gfCNCPoint5[10865] = {X 236.2309, Y 48.3200, Z -7.1667, A 0.000, B 0.000, C 0.000 }
gfCNCPoint5[10866] = {X 235.6245, Y 47.5134, Z -7.1667, A 0.000, B 0.000, C 0.000 }
gfCNCPoint5[10867] = {X 235.1970, Y 46.5992, Z -7.1667, A 0.000, B 0.000, C 0.000 }
gfCNCPoint5[10868] = {X 234.9666, Y 45.6167, Z -7.1667, A 0.000, B 0.000, C 0.000 }
gfCNCPoint5[10869] = {X 234.9373, Y 45.3090, Z -7.1667, A 0.000, B 0.000, C 0.000 }
gfCNCPoint5[10870] = {X 234.9275, Y 45.0000, Z -7.1667, A 0.000, B 0.000, C 0.000 }
gfCNCPoint5[10871] = {X 234.9275, Y 44.2089, Z -7.1667, A 0.000, B 0.000, C 0.000 }
gfCNCPoint5[10872] = {X 235.0194, Y 43.2661, Z -7.1667, A 0.000, B 0.000, C 0.000 }
gfCNCPoint5[10873] = {X 235.2918, Y 42.3588, Z -7.1667, A 0.000, B 0.000, C 0.000 }
gfCNCPoint5[10874] = {X 235.7342, Y 41.5212, Z -7.1667, A 0.000, B 0.000, C 0.000 }
gfCNCPoint5[10875] = {X 236.3302, Y 40.7849, Z -7.1667, A 0.000, B 0.000, C 0.000 }
gfCNCPoint5[10876] = {X 237.0572, Y 40.1776, Z -7.1667, A 0.000, B 0.000, C 0.000 }
gfCNCPoint5[10877] = {X 237.8878, Y 39.7222, Z -7.1667, A 0.000, B 0.000, C 0.000 }
gfCNCPoint5[10878] = {X 241.5460, Y 32.5618, Z -7.1667, A 0.000, B 0.000, C 0.000 }
gfCNCPoint5[10879] = {X 240.2114, Y 31.5589, Z -7.1667, A 0.000, B 0.000, C 0.000 }
gfCNCPoint5[10880] = {X 239.0306, Y 30.3788, Z -7.1667, A 0.000, B 0.000, C 0.000 }
gfCNCPoint5[10881] = {X 238.0268, Y 29.0450, Z -7.1667, A 0.000, B 0.000, C 0.000 }
gfCNCPoint5[10882] = {X 237.2198, Y 27.5836, Z -7.1667, A 0.000, B 0.000, C 0.000 }
gfCNCPoint5[10883] = {X 236.6256, Y 26.0236, Z -7.1667, A 0.000, B 0.000, C 0.000 }
gfCNCPoint5[10884] = {X 236.1904, Y 24.1499, Z -7.1667, A 0.000, B 0.000, C 0.000 }
gfCNCPoint5[10885] = {X 235.9685, Y 22.2393, Z -7.1667, A 0.000, B 0.000, C 0.000 }
gfCNCPoint5[10886] = {X 235.9626, Y 20.3158, Z -7.1667, A 0.000, B 0.000, C 0.000 }
gfCNCPoint5[10887] = {X 236.1729, Y 18.4038, Z -7.1667, A 0.000, B 0.000, C 0.000 }
gfCNCPoint5[10888] = {X 236.5966, Y 16.5276, Z -7.1667, A 0.000, B 0.000, C 0.000 }
gfCNCPoint5[10889] = {X 237.1160, Y 15.0570, Z -7.1667, A 0.000, B 0.000, C 0.000 }
gfCNCPoint5[10890] = {X 237.8157, Y 13.6631, Z -7.1667, A 0.000, B 0.000, C 0.000 }
gfCNCPoint5[10891] = {X 238.6848, Y 12.3680, Z -7.1667, A 0.000, B 0.000, C 0.000 }
gfCNCPoint5[10892] = {X 239.7094, Y 11.1921, Z -7.1667, A 0.000, B 0.000, C 0.000 }
gfCNCPoint5[10893] = {X 240.8738, Y 10.1538, Z -7.1667, A 0.000, B 0.000, C 0.000 }
gfCNCPoint5[10894] = {X 242.1593, Y 9.2697, Z -7.1667, A 0.000, B 0.000, C 0.000 }
gfCNCPoint5[10895] = {X 243.5456, Y 8.5539, Z -7.1667, A 0.000, B 0.000, C 0.000 }
gfCNCPoint5[10896] = {X 245.0107, Y 8.0176, Z -7.1667, A 0.000, B 0.000, C 0.000 }
gfCNCPoint5[10897] = {X 246.5316, Y 7.6695, Z -7.1667, A 0.000, B 0.000, C 0.000 }
gfCNCPoint5[10898] = {X 248.6761, Y 7.3920, Z -7.1667, A 0.000, B 0.000, C 0.000 }
gfCNCPoint5[10899] = {X 250.8369, Y 7.3096, Z -7.1667, A 0.000, B 0.000, C 0.000 }
gfCNCPoint5[10900] = {X 266.7608, Y 7.3096, Z -7.1667, A 0.000, B 0.000, C 0.000 }
gfCNCPoint5[10901] = {X 267.7192, Y 7.4110, Z -7.1667, A 0.000, B 0.000, C 0.000 }
gfCNCPoint5[10902] = {X 268.6390, Y 7.6987, Z -7.1667, A 0.000, B 0.000, C 0.000 }
gfCNCPoint5[10903] = {X 269.4844, Y 8.1615, Z -7.1667, A 0.000, B 0.000, C 0.000 }
gfCNCPoint5[10904] = {X 270.2224, Y 8.7814, Z -7.1667, A 0.000, B 0.000, C 0.000 }
gfCNCPoint5[10905] = {X 270.8243, Y 9.5341, Z -7.1667, A 0.000, B 0.000, C 0.000 }
gfCNCPoint5[10906] = {X 271.2665, Y 10.3904, Z -7.1667, A 0.000, B 0.000, C 0.000 }
gfCNCPoint5[10907] = {X 271.5236, Y 11.2718, Z -7.1667, A 0.000, B 0.000, C 0.000 }
gfCNCPoint5[10908] = {X 271.6110, Y 12.1858, Z -7.1667, A 0.000, B 0.000, C 0.000 }
gfCNCPoint5[10909] = {X 271.6108, Y 13.0237, Z -7.1667, A 0.000, B 0.000, C 0.000 }
gfCNCPoint5[10910] = {X 271.5128, Y 13.9524, Z -7.1667, A 0.000, B 0.000, C 0.000 }
gfCNCPoint5[10911] = {X 271.2396, Y 14.8453, Z -7.1667, A 0.000, B 0.000, C 0.000 }
gfCNCPoint5[10912] = {X 275.6743, Y 16.6820, Z -7.1667, A 0.000, B 0.000, C 0.000 }
gfCNCPoint5[10913] = {X 275.3129, Y 17.4561, Z -7.1667, A 0.000, B 0.000, C 0.000 }
gfCNCPoint5[10914] = {X 274.8847, Y 18.1954, Z -7.1667, A 0.000, B 0.000, C 0.000 }
gfCNCPoint5[10915] = {X 274.8848, Y 38.9916, Z -7.1667, A 0.000, B 0.000, C 0.000 }
gfCNCPoint5[10916] = {X 275.3141, Y 39.7329, Z -7.1667, A 0.000, B 0.000, C 0.000 }
gfCNCPoint5[10917] = {X 275.6762, Y 40.5092, Z -7.1667, A 0.000, B 0.000, C 0.000 }
gfCNCPoint5[10918] = {X 276.0370, Y 39.7351, Z -7.1667, A 0.000, B 0.000, C 0.000 }
gfCNCPoint5[10919] = {X 276.4644, Y 38.9955, Z -7.1667, A 0.000, B 0.000, C 0.000 }
gfCNCPoint5[10920] = {X 276.4643, Y 18.1958, Z -7.1667, A 0.000, B 0.000, C 0.000 }
gfCNCPoint5[10921] = {X 276.0359, Y 17.4563, Z -7.1667, A 0.000, B 0.000, C 0.000 }
gfCNCPoint5[10922] = {X 275.6743, Y 16.6820, Z -7.1667, A 0.000, B 0.000, C 0.000 }
gfCNCPoint5[10923] = {X 273.4570, Y 15.7637, Z -7.1667, A 0.000, B 0.000, C 0.000 }
gfCNCPoint5[10924] = {X 273.0268, Y 16.6335, Z -7.1667, A 0.000, B 0.000, C 0.000 }
gfCNCPoint5[10925] = {X 272.4847, Y 17.4383, Z -7.1667, A 0.000, B 0.000, C 0.000 }
gfCNCPoint5[10926] = {X 272.4848, Y 39.7486, Z -7.1667, A 0.000, B 0.000, C 0.000 }
gfCNCPoint5[10927] = {X 273.0277, Y 40.5550, Z -7.1667, A 0.000, B 0.000, C 0.000 }
gfCNCPoint5[10928] = {X 273.4584, Y 41.4265, Z -7.1667, A 0.000, B 0.000, C 0.000 }
gfCNCPoint5[10929] = {X 273.7587, Y 42.3088, Z -7.1667, A 0.000, B 0.000, C 0.000 }
gfCNCPoint5[10930] = {X 273.9439, Y 43.2222, Z -7.1667, A 0.000, B 0.000, C 0.000 }
gfCNCPoint5[10931] = {X 274.0108, Y 44.1519, Z -7.1667, A 0.000, B 0.000, C 0.000 }
gfCNCPoint5[10932] = {X 274.0110, Y 45.0000, Z -7.1667, A 0.000, B 0.000, C 0.000 }
gfCNCPoint5[10933] = {X 273.9884, Y 45.5734, Z -7.1667, A 0.000, B 0.000, C 0.000 }
gfCNCPoint5[10934] = {X 273.9207, Y 46.1433, Z -7.1667, A 0.000, B 0.000, C 0.000 }
gfCNCPoint5[10935] = {X 275.0713, Y 45.9760, Z -7.1667, A 0.000, B 0.000, C 0.000 }
gfCNCPoint5[10936] = {X 276.2327, Y 45.9200, Z -7.1667, A 0.000, B 0.000, C 0.000 }
gfCNCPoint5[10937] = {X 277.3960, Y 45.9200, Z -7.1667, A 0.000, B 0.000, C 0.000 }
gfCNCPoint5[10938] = {X 277.3539, Y 45.4858, Z -7.1667, A 0.000, B 0.000, C 0.000 }
gfCNCPoint5[10939] = {X 277.3378, Y 45.0498, Z -7.1667, A 0.000, B 0.000, C 0.000 }
gfCNCPoint5[10940] = {X 277.3377, Y 44.2000, Z -7.1667, A 0.000, B 0.000, C 0.000 }
gfCNCPoint5[10941] = {X 277.4025, Y 43.2541, Z -7.1667, A 0.000, B 0.000, C 0.000 }
gfCNCPoint5[10942] = {X 277.5889, Y 42.3244, Z -7.1667, A 0.000, B 0.000, C 0.000 }
gfCNCPoint5[10943] = {X 277.8939, Y 41.4266, Z -7.1667, A 0.000, B 0.000, C 0.000 }
gfCNCPoint5[10944] = {X 278.3235, Y 40.5564, Z -7.1667, A 0.000, B 0.000, C 0.000 }
gfCNCPoint5[10945] = {X 278.8644, Y 39.7505, Z -7.1667, A 0.000, B 0.000, C 0.000 }
gfCNCPoint5[10946] = {X 278.8643, Y 17.4386, Z -7.1667, A 0.000, B 0.000, C 0.000 }
gfCNCPoint5[10947] = {X 278.3220, Y 16.6336, Z -7.1667, A 0.000, B 0.000, C 0.000 }
gfCNCPoint5[10948] = {X 277.8917, Y 15.7637, Z -7.1667, A 0.000, B 0.000, C 0.000 }
gfCNCPoint5[10949] = {X 277.5902, Y 14.8788, Z -7.1667, A 0.000, B 0.000, C 0.000 }
gfCNCPoint5[10950] = {X 277.4046, Y 13.9627, Z -7.1667, A 0.000, B 0.000, C 0.000 }
gfCNCPoint5[10951] = {X 277.3379, Y 13.0303, Z -7.1667, A 0.000, B 0.000, C 0.000 }
gfCNCPoint5[10952] = {X 277.3377, Y 12.1868, Z -7.1667, A 0.000, B 0.000, C 0.000 }
gfCNCPoint5[10953] = {X 277.3952, Y 11.2737, Z -7.1667, A 0.000, B 0.000, C 0.000 }
gfCNCPoint5[10954] = {X 277.5667, Y 10.3750, Z -7.1667, A 0.000, B 0.000, C 0.000 }
gfCNCPoint5[10955] = {X 277.8497, Y 9.5049, Z -7.1667, A 0.000, B 0.000, C 0.000 }
gfCNCPoint5[10956] = {X 273.4972, Y 9.5049, Z -7.1667, A 0.000, B 0.000, C 0.000 }
gfCNCPoint5[10957] = {X 273.7804, Y 10.3736, Z -7.1667, A 0.000, B 0.000, C 0.000 }
gfCNCPoint5[10958] = {X 273.9526, Y 11.2709, Z -7.1667, A 0.000, B 0.000, C 0.000 }
gfCNCPoint5[10959] = {X 274.0110, Y 12.1828, Z -7.1667, A 0.000, B 0.000, C 0.000 }
gfCNCPoint5[10960] = {X 274.0107, Y 13.0462, Z -7.1667, A 0.000, B 0.000, C 0.000 }
gfCNCPoint5[10961] = {X 273.9427, Y 13.9732, Z -7.1667, A 0.000, B 0.000, C 0.000 }
gfCNCPoint5[10962] = {X 273.7571, Y 14.8840, Z -7.1667, A 0.000, B 0.000, C 0.000 }
gfCNCPoint5[10963] = {X 273.4570, Y 15.7637, Z -7.1667, A 0.000, B 0.000, C 0.000 }
gfCNCPoint5[10964] = {X 271.2396, Y 14.8453, Z -7.1667, A 0.000, B 0.000, C 0.000 }
gfCNCPoint5[10965] = {X 270.7507, Y 15.7451, Z -7.1667, A 0.000, B 0.000, C 0.000 }
gfCNCPoint5[10966] = {X 270.0847, Y 16.5231, Z -7.1667, A 0.000, B 0.000, C 0.000 }
gfCNCPoint5[10967] = {X 270.0848, Y 40.6638, Z -7.1667, A 0.000, B 0.000, C 0.000 }
gfCNCPoint5[10968] = {X 270.7249, Y 41.4045, Z -7.1667, A 0.000, B 0.000, C 0.000 }
gfCNCPoint5[10969] = {X 271.2042, Y 42.2581, Z -7.1667, A 0.000, B 0.000, C 0.000 }
gfCNCPoint5[10970] = {X 271.5036, Y 43.1902, Z -7.1667, A 0.000, B 0.000, C 0.000 }
gfCNCPoint5[10971] = {X 271.6108, Y 44.1633, Z -7.1667, A 0.000, B 0.000, C 0.000 }
gfCNCPoint5[10972] = {X 271.6110, Y 45.0000, Z -7.1667, A 0.000, B 0.000, C 0.000 }
gfCNCPoint5[10973] = {X 271.5959, Y 45.3844, Z -7.1667, A 0.000, B 0.000, C 0.000 }
gfCNCPoint5[10974] = {X 271.5505, Y 45.7664, Z -7.1667, A 0.000, B 0.000, C 0.000 }
gfCNCPoint5[10975] = {X 271.2989, Y 46.7171, Z -7.1667, A 0.000, B 0.000, C 0.000 }
gfCNCPoint5[10976] = {X 270.8619, Y 47.5982, Z -7.1667, A 0.000, B 0.000, C 0.000 }
gfCNCPoint5[10977] = {X 270.2571, Y 48.3736, Z -7.1667, A 0.000, B 0.000, C 0.000 }
gfCNCPoint5[10978] = {X 269.5090, Y 49.0121, Z -7.1667, A 0.000, B 0.000, C 0.000 }
gfCNCPoint5[10979] = {X 268.6482, Y 49.4876, Z -7.1667, A 0.000, B 0.000, C 0.000 }
gfCNCPoint5[10980] = {X 267.7095, Y 49.7809, Z -7.1667, A 0.000, B 0.000, C 0.000 }
gfCNCPoint5[10981] = {X 266.7310, Y 49.8800, Z -7.1667, A 0.000, B 0.000, C 0.000 }
gfCNCPoint5[10982] = {X 262.1384, Y 49.8800, Z -7.1667, A 0.000, B 0.000, C 0.000 }
gfCNCPoint5[10983] = {X 262.1384, Y 54.6800, Z -7.1667, A 0.000, B 0.000, C 0.000 }
gfCNCPoint5[10984] = {X 260.2880, Y 54.6800, Z -7.1667, A 0.000, B 0.000, C 0.000 }
gfCNCPoint5[10985] = {X 261.9958, Y 55.3579, Z -7.1667, A 0.000, B 0.000, C 0.000 }
gfCNCPoint5[10986] = {X 262.0631, Y 55.0181, Z -7.1667, A 0.000, B 0.000, C 0.000 }
gfCNCPoint5[10987] = {X 262.1384, Y 54.6800, Z -7.1667, A 0.000, B 0.000, C 0.000 }
gfCNCPoint5[10988] = {X 262.1384, Y 52.2800, Z -7.1667, A 0.000, B 0.000, C 0.000 }
gfCNCPoint5[10989] = {X 260.2876, Y 52.2800, Z -7.1667, A 0.000, B 0.000, C 0.000 }
gfCNCPoint5[10990] = {X 259.1914, Y 52.1970, Z -7.1667, A 0.000, B 0.000, C 0.000 }
gfCNCPoint5[10991] = {X 258.1202, Y 51.9499, Z -7.1667, A 0.000, B 0.000, C 0.000 }
gfCNCPoint5[10992] = {X 257.0985, Y 51.5443, Z -7.1667, A 0.000, B 0.000, C 0.000 }
gfCNCPoint5[10993] = {X 256.1494, Y 50.9895, Z -7.1667, A 0.000, B 0.000, C 0.000 }
gfCNCPoint5[10994] = {X 255.2947, Y 50.2981, Z -7.1667, A 0.000, B 0.000, C 0.000 }
gfCNCPoint5[10995] = {X 253.6488, Y 52.0448, Z -7.1667, A 0.000, B 0.000, C 0.000 }
gfCNCPoint5[10996] = {X 253.4930, Y 51.8946, Z -7.1667, A 0.000, B 0.000, C 0.000 }
gfCNCPoint5[10997] = {X 253.3406, Y 51.7410, Z -7.1667, A 0.000, B 0.000, C 0.000 }
gfCNCPoint5[10998] = {X 253.2765, Y 51.8065, Z -7.1667, A 0.000, B 0.000, C 0.000 }
gfCNCPoint5[10999] = {X 253.2117, Y 51.8713, Z -7.1667, A 0.000, B 0.000, C 0.000 }
gfCNCPoint5[11000] = {X 253.6488, Y 52.0448, Z -7.1667, A 0.000, B 0.000, C 0.000 }
gfCNCPoint5[11001] = {X 255.2947, Y 50.2981, Z -7.1667, A 0.000, B 0.000, C 0.000 }
gfCNCPoint5[11002] = {X 255.1776, Y 50.1852, Z -7.1667, A 0.000, B 0.000, C 0.000 }
gfCNCPoint5[11003] = {X 255.0630, Y 50.0697, Z -7.1667, A 0.000, B 0.000, C 0.000 }
gfCNCPoint5[11004] = {X 254.3405, Y 49.1989, Z -7.1667, A 0.000, B 0.000, C 0.000 }
gfCNCPoint5[11005] = {X 253.7617, Y 48.2267, Z -7.1667, A 0.000, B 0.000, C 0.000 }
gfCNCPoint5[11006] = {X 253.3406, Y 47.1766, Z -7.1667, A 0.000, B 0.000, C 0.000 }
gfCNCPoint5[11007] = {X 252.9194, Y 48.2267, Z -7.1667, A 0.000, B 0.000, C 0.000 }
gfCNCPoint5[11008] = {X 252.3406, Y 49.1989, Z -7.1667, A 0.000, B 0.000, C 0.000 }
gfCNCPoint5[11009] = {X 251.6182, Y 50.0697, Z -7.1667, A 0.000, B 0.000, C 0.000 }
gfCNCPoint5[11010] = {X 251.5700, Y 50.1189, Z -7.1667, A 0.000, B 0.000, C 0.000 }
gfCNCPoint5[11011] = {X 251.5213, Y 50.1677, Z -7.1667, A 0.000, B 0.000, C 0.000 }
gfCNCPoint5[11012] = {X 250.7153, Y 50.8584, Z -7.1667, A 0.000, B 0.000, C 0.000 }
gfCNCPoint5[11013] = {X 249.8175, Y 51.4246, Z -7.1667, A 0.000, B 0.000, C 0.000 }
gfCNCPoint5[11014] = {X 248.8469, Y 51.8542, Z -7.1667, A 0.000, B 0.000, C 0.000 }
gfCNCPoint5[11015] = {X 247.8241, Y 52.1381, Z -7.1667, A 0.000, B 0.000, C 0.000 }
gfCNCPoint5[11016] = {X 247.8927, Y 52.2635, Z -7.1667, A 0.000, B 0.000, C 0.000 }
gfCNCPoint5[11017] = {X 247.9599, Y 52.3898, Z -7.1667, A 0.000, B 0.000, C 0.000 }
gfCNCPoint5[11018] = {X 250.9688, Y 53.5632, Z -7.1667, A 0.000, B 0.000, C 0.000 }
gfCNCPoint5[11019] = {X 264.1528, Y 58.7962, Z -7.1667, A 0.000, B 0.000, C 0.000 }
gfCNCPoint5[11020] = {X 264.1527, Y 58.0000, Z -7.1667, A 0.000, B 0.000, C 0.000 }
gfCNCPoint5[11021] = {X 264.2035, Y 56.8932, Z -7.1667, A 0.000, B 0.000, C 0.000 }
gfCNCPoint5[11022] = {X 264.3555, Y 55.7958, Z -7.1667, A 0.000, B 0.000, C 0.000 }
gfCNCPoint5[11023] = {X 264.4116, Y 55.5123, Z -7.1667, A 0.000, B 0.000, C 0.000 }
gfCNCPoint5[11024] = {X 264.4745, Y 55.2303, Z -7.1667, A 0.000, B 0.000, C 0.000 }
gfCNCPoint5[11025] = {X 264.9369, Y 53.7185, Z -7.1667, A 0.000, B 0.000, C 0.000 }
gfCNCPoint5[11026] = {X 265.5928, Y 52.2800, Z -7.1667, A 0.000, B 0.000, C 0.000 }
gfCNCPoint5[11027] = {X 262.1384, Y 52.2800, Z -7.1667, A 0.000, B 0.000, C 0.000 }
gfCNCPoint5[11028] = {X 262.1384, Y 49.8800, Z -7.1667, A 0.000, B 0.000, C 0.000 }
gfCNCPoint5[11029] = {X 260.2876, Y 49.8800, Z -7.1667, A 0.000, B 0.000, C 0.000 }
gfCNCPoint5[11030] = {X 259.2646, Y 49.7716, Z -7.1667, A 0.000, B 0.000, C 0.000 }
gfCNCPoint5[11031] = {X 258.2870, Y 49.4511, Z -7.1667, A 0.000, B 0.000, C 0.000 }
gfCNCPoint5[11032] = {X 257.3984, Y 48.9328, Z -7.1667, A 0.000, B 0.000, C 0.000 }
gfCNCPoint5[11033] = {X 256.6382, Y 48.2398, Z -7.1667, A 0.000, B 0.000, C 0.000 }
gfCNCPoint5[11034] = {X 256.0401, Y 47.4028, Z -7.1667, A 0.000, B 0.000, C 0.000 }
gfCNCPoint5[11035] = {X 255.6308, Y 46.4590, Z -7.1667, A 0.000, B 0.000, C 0.000 }
gfCNCPoint5[11036] = {X 255.4666, Y 45.7568, Z -7.1667, A 0.000, B 0.000, C 0.000 }
gfCNCPoint5[11037] = {X 255.4077, Y 45.0380, Z -7.1667, A 0.000, B 0.000, C 0.000 }
gfCNCPoint5[11038] = {X 255.4080, Y 44.1417, Z -7.1667, A 0.000, B 0.000, C 0.000 }
gfCNCPoint5[11039] = {X 255.5183, Y 43.1751, Z -7.1667, A 0.000, B 0.000, C 0.000 }
gfCNCPoint5[11040] = {X 255.8181, Y 42.2497, Z -7.1667, A 0.000, B 0.000, C 0.000 }
gfCNCPoint5[11041] = {X 256.2955, Y 41.4021, Z -7.1667, A 0.000, B 0.000, C 0.000 }
gfCNCPoint5[11042] = {X 256.9315, Y 40.6660, Z -7.1667, A 0.000, B 0.000, C 0.000 }
gfCNCPoint5[11043] = {X 256.9315, Y 35.0338, Z -7.1667, A 0.000, B 0.000, C 0.000 }
gfCNCPoint5[11044] = {X 255.1106, Y 35.0338, Z -7.1667, A 0.000, B 0.000, C 0.000 }
gfCNCPoint5[11045] = {X 251.0867, Y 42.8714, Z -7.1667, A 0.000, B 0.000, C 0.000 }
gfCNCPoint5[11046] = {X 251.2237, Y 43.5132, Z -7.1667, A 0.000, B 0.000, C 0.000 }
gfCNCPoint5[11047] = {X 251.2734, Y 44.1675, Z -7.1667, A 0.000, B 0.000, C 0.000 }
gfCNCPoint5[11048] = {X 251.2736, Y 45.0000, Z -7.1667, A 0.000, B 0.000, C 0.000 }
gfCNCPoint5[11049] = {X 251.2174, Y 45.7380, Z -7.1667, A 0.000, B 0.000, C 0.000 }
gfCNCPoint5[11050] = {X 251.0503, Y 46.4590, Z -7.1667, A 0.000, B 0.000, C 0.000 }
gfCNCPoint5[11051] = {X 250.6346, Y 47.4142, Z -7.1667, A 0.000, B 0.000, C 0.000 }
gfCNCPoint5[11052] = {X 250.0255, Y 48.2593, Z -7.1667, A 0.000, B 0.000, C 0.000 }
gfCNCPoint5[11053] = {X 249.2510, Y 48.9560, Z -7.1667, A 0.000, B 0.000, C 0.000 }
gfCNCPoint5[11054] = {X 248.3462, Y 49.4723, Z -7.1667, A 0.000, B 0.000, C 0.000 }
gfCNCPoint5[11055] = {X 247.3525, Y 49.7849, Z -7.1667, A 0.000, B 0.000, C 0.000 }
gfCNCPoint5[11056] = {X 246.8754, Y 49.8562, Z -7.1667, A 0.000, B 0.000, C 0.000 }
gfCNCPoint5[11057] = {X 246.3936, Y 49.8800, Z -7.1667, A 0.000, B 0.000, C 0.000 }
gfCNCPoint5[11058] = {X 242.5312, Y 49.8800, Z -7.1667, A 0.000, B 0.000, C 0.000 }
gfCNCPoint5[11059] = {X 242.5312, Y 49.4000, Z -7.1667, A 0.000, B 0.000, C 0.000 }
gfCNCPoint5[11060] = {X 239.8075, Y 49.4000, Z -7.1667, A 0.000, B 0.000, C 0.000 }
gfCNCPoint5[11061] = {X 238.8284, Y 49.2897, Z -7.1667, A 0.000, B 0.000, C 0.000 }
gfCNCPoint5[11062] = {X 237.8984, Y 48.9643, Z -7.1667, A 0.000, B 0.000, C 0.000 }
gfCNCPoint5[11063] = {X 237.0641, Y 48.4401, Z -7.1667, A 0.000, B 0.000, C 0.000 }
gfCNCPoint5[11064] = {X 236.3674, Y 47.7434, Z -7.1667, A 0.000, B 0.000, C 0.000 }
gfCNCPoint5[11065] = {X 235.8432, Y 46.9091, Z -7.1667, A 0.000, B 0.000, C 0.000 }
gfCNCPoint5[11066] = {X 235.5178, Y 45.9791, Z -7.1667, A 0.000, B 0.000, C 0.000 }
gfCNCPoint5[11067] = {X 235.4075, Y 45.0000, Z -7.1667, A 0.000, B 0.000, C 0.000 }
gfCNCPoint5[11068] = {X 235.4079, Y 44.1483, Z -7.1667, A 0.000, B 0.000, C 0.000 }
gfCNCPoint5[11069] = {X 235.5063, Y 43.2816, Z -7.1667, A 0.000, B 0.000, C 0.000 }
gfCNCPoint5[11070] = {X 235.7737, Y 42.4514, Z -7.1667, A 0.000, B 0.000, C 0.000 }
gfCNCPoint5[11071] = {X 236.1996, Y 41.6903, Z -7.1667, A 0.000, B 0.000, C 0.000 }
gfCNCPoint5[11072] = {X 236.7672, Y 41.0281, Z -7.1667, A 0.000, B 0.000, C 0.000 }
gfCNCPoint5[11073] = {X 237.4544, Y 40.4909, Z -7.1667, A 0.000, B 0.000, C 0.000 }
gfCNCPoint5[11074] = {X 238.2339, Y 40.0998, Z -7.1667, A 0.000, B 0.000, C 0.000 }
gfCNCPoint5[11075] = {X 242.1744, Y 32.3868, Z -7.1667, A 0.000, B 0.000, C 0.000 }
gfCNCPoint5[11076] = {X 241.0108, Y 31.5942, Z -7.1667, A 0.000, B 0.000, C 0.000 }
gfCNCPoint5[11077] = {X 239.9537, Y 30.6642, Z -7.1667, A 0.000, B 0.000, C 0.000 }
gfCNCPoint5[11078] = {X 239.0193, Y 29.6110, Z -7.1667, A 0.000, B 0.000, C 0.000 }
gfCNCPoint5[11079] = {X 238.2218, Y 28.4508, Z -7.1667, A 0.000, B 0.000, C 0.000 }
gfCNCPoint5[11080] = {X 237.5734, Y 27.2010, Z -7.1667, A 0.000, B 0.000, C 0.000 }
gfCNCPoint5[11081] = {X 237.0839, Y 25.8809, Z -7.1667, A 0.000, B 0.000, C 0.000 }
gfCNCPoint5[11082] = {X 236.6622, Y 24.0613, Z -7.1667, A 0.000, B 0.000, C 0.000 }
gfCNCPoint5[11083] = {X 236.4473, Y 22.2057, Z -7.1667, A 0.000, B 0.000, C 0.000 }
gfCNCPoint5[11084] = {X 236.4421, Y 20.3378, Z -7.1667, A 0.000, B 0.000, C 0.000 }
gfCNCPoint5[11085] = {X 236.6466, Y 18.4811, Z -7.1667, A 0.000, B 0.000, C 0.000 }
gfCNCPoint5[11086] = {X 237.0582, Y 16.6591, Z -7.1667, A 0.000, B 0.000, C 0.000 }
gfCNCPoint5[11087] = {X 237.6326, Y 15.0727, Z -7.1667, A 0.000, B 0.000, C 0.000 }
gfCNCPoint5[11088] = {X 238.4250, Y 13.5832, Z -7.1667, A 0.000, B 0.000, C 0.000 }
gfCNCPoint5[11089] = {X 239.4195, Y 12.2203, Z -7.1667, A 0.000, B 0.000, C 0.000 }
gfCNCPoint5[11090] = {X 240.5964, Y 11.0114, Z -7.1667, A 0.000, B 0.000, C 0.000 }
gfCNCPoint5[11091] = {X 241.9321, Y 9.9806, Z -7.1667, A 0.000, B 0.000, C 0.000 }
gfCNCPoint5[11092] = {X 243.3998, Y 9.1485, Z -7.1667, A 0.000, B 0.000, C 0.000 }
gfCNCPoint5[11093] = {X 244.9702, Y 8.5318, Z -7.1667, A 0.000, B 0.000, C 0.000 }
gfCNCPoint5[11094] = {X 246.6119, Y 8.1427, Z -7.1667, A 0.000, B 0.000, C 0.000 }
gfCNCPoint5[11095] = {X 248.7155, Y 7.8704, Z -7.1667, A 0.000, B 0.000, C 0.000 }
gfCNCPoint5[11096] = {X 250.8351, Y 7.7896, Z -7.1667, A 0.000, B 0.000, C 0.000 }
gfCNCPoint5[11097] = {X 266.7640, Y 7.7896, Z -7.1667, A 0.000, B 0.000, C 0.000 }
gfCNCPoint5[11098] = {X 267.7370, Y 7.9065, Z -7.1667, A 0.000, B 0.000, C 0.000 }
gfCNCPoint5[11099] = {X 268.6601, Y 8.2357, Z -7.1667, A 0.000, B 0.000, C 0.000 }
gfCNCPoint5[11100] = {X 269.4874, Y 8.7610, Z -7.1667, A 0.000, B 0.000, C 0.000 }
gfCNCPoint5[11101] = {X 270.1781, Y 9.4564, Z -7.1667, A 0.000, B 0.000, C 0.000 }
gfCNCPoint5[11102] = {X 270.6977, Y 10.2873, Z -7.1667, A 0.000, B 0.000, C 0.000 }
gfCNCPoint5[11103] = {X 271.0207, Y 11.2125, Z -7.1667, A 0.000, B 0.000, C 0.000 }
gfCNCPoint5[11104] = {X 271.1310, Y 12.1864, Z -7.1667, A 0.000, B 0.000, C 0.000 }
gfCNCPoint5[11105] = {X 271.1308, Y 13.0233, Z -7.1667, A 0.000, B 0.000, C 0.000 }
gfCNCPoint5[11106] = {X 271.0226, Y 13.9490, Z -7.1667, A 0.000, B 0.000, C 0.000 }
gfCNCPoint5[11107] = {X 270.7218, Y 14.8311, Z -7.1667, A 0.000, B 0.000, C 0.000 }
gfCNCPoint5[11108] = {X 270.2420, Y 15.6300, Z -7.1667, A 0.000, B 0.000, C 0.000 }
gfCNCPoint5[11109] = {X 269.6047, Y 16.3100, Z -7.1667, A 0.000, B 0.000, C 0.000 }
gfCNCPoint5[11110] = {X 269.6048, Y 40.8769, Z -7.1667, A 0.000, B 0.000, C 0.000 }
gfCNCPoint5[11111] = {X 270.2489, Y 41.5659, Z -7.1667, A 0.000, B 0.000, C 0.000 }
gfCNCPoint5[11112] = {X 270.7313, Y 42.3764, Z -7.1667, A 0.000, B 0.000, C 0.000 }
gfCNCPoint5[11113] = {X 271.0300, Y 43.2711, Z -7.1667, A 0.000, B 0.000, C 0.000 }
gfCNCPoint5[11114] = {X 271.1310, Y 44.2089, Z -7.1667, A 0.000, B 0.000, C 0.000 }
gfCNCPoint5[11115] = {X 271.1310, Y 45.0000, Z -7.1667, A 0.000, B 0.000, C 0.000 }
gfCNCPoint5[11116] = {X 271.0207, Y 45.9791, Z -7.1667, A 0.000, B 0.000, C 0.000 }
gfCNCPoint5[11117] = {X 270.6953, Y 46.9091, Z -7.1667, A 0.000, B 0.000, C 0.000 }
gfCNCPoint5[11118] = {X 270.1711, Y 47.7434, Z -7.1667, A 0.000, B 0.000, C 0.000 }
gfCNCPoint5[11119] = {X 269.4744, Y 48.4401, Z -7.1667, A 0.000, B 0.000, C 0.000 }
gfCNCPoint5[11120] = {X 268.6401, Y 48.9643, Z -7.1667, A 0.000, B 0.000, C 0.000 }
gfCNCPoint5[11121] = {X 267.7101, Y 49.2897, Z -7.1667, A 0.000, B 0.000, C 0.000 }
gfCNCPoint5[11122] = {X 266.7310, Y 49.4000, Z -7.1667, A 0.000, B 0.000, C 0.000 }
gfCNCPoint5[11123] = {X 260.2876, Y 49.4000, Z -7.1667, A 0.000, B 0.000, C 0.000 }
gfCNCPoint5[11124] = {X 259.3085, Y 49.2897, Z -7.1667, A 0.000, B 0.000, C 0.000 }
gfCNCPoint5[11125] = {X 258.3785, Y 48.9643, Z -7.1667, A 0.000, B 0.000, C 0.000 }
gfCNCPoint5[11126] = {X 257.5442, Y 48.4401, Z -7.1667, A 0.000, B 0.000, C 0.000 }
gfCNCPoint5[11127] = {X 256.8475, Y 47.7433, Z -7.1667, A 0.000, B 0.000, C 0.000 }
gfCNCPoint5[11128] = {X 256.3233, Y 46.9091, Z -7.1667, A 0.000, B 0.000, C 0.000 }
gfCNCPoint5[11129] = {X 255.9979, Y 45.9791, Z -7.1667, A 0.000, B 0.000, C 0.000 }
gfCNCPoint5[11130] = {X 255.8876, Y 45.0000, Z -7.1667, A 0.000, B 0.000, C 0.000 }
gfCNCPoint5[11131] = {X 255.8880, Y 44.1483, Z -7.1667, A 0.000, B 0.000, C 0.000 }
gfCNCPoint5[11132] = {X 255.9984, Y 43.2275, Z -7.1667, A 0.000, B 0.000, C 0.000 }
gfCNCPoint5[11133] = {X 256.2993, Y 42.3503, Z -7.1667, A 0.000, B 0.000, C 0.000 }
gfCNCPoint5[11134] = {X 256.7775, Y 41.5556, Z -7.1667, A 0.000, B 0.000, C 0.000 }
gfCNCPoint5[11135] = {X 257.4115, Y 40.8789, Z -7.1667, A 0.000, B 0.000, C 0.000 }
gfCNCPoint5[11136] = {X 257.4115, Y 34.5538, Z -7.1667, A 0.000, B 0.000, C 0.000 }
gfCNCPoint5[11137] = {X 254.8175, Y 34.5538, Z -7.1667, A 0.000, B 0.000, C 0.000 }
gfCNCPoint5[11138] = {X 250.5706, Y 42.8258, Z -7.1667, A 0.000, B 0.000, C 0.000 }
gfCNCPoint5[11139] = {X 250.7375, Y 43.5084, Z -7.1667, A 0.000, B 0.000, C 0.000 }
gfCNCPoint5[11140] = {X 250.7936, Y 44.2089, Z -7.1667, A 0.000, B 0.000, C 0.000 }
gfCNCPoint5[11141] = {X 250.7936, Y 45.0000, Z -7.1667, A 0.000, B 0.000, C 0.000 }
gfCNCPoint5[11142] = {X 250.6832, Y 45.9791, Z -7.1667, A 0.000, B 0.000, C 0.000 }
gfCNCPoint5[11143] = {X 250.3578, Y 46.9091, Z -7.1667, A 0.000, B 0.000, C 0.000 }
gfCNCPoint5[11144] = {X 249.8336, Y 47.7434, Z -7.1667, A 0.000, B 0.000, C 0.000 }
gfCNCPoint5[11145] = {X 249.1369, Y 48.4401, Z -7.1667, A 0.000, B 0.000, C 0.000 }
gfCNCPoint5[11146] = {X 248.3026, Y 48.9643, Z -7.1667, A 0.000, B 0.000, C 0.000 }
gfCNCPoint5[11147] = {X 247.3727, Y 49.2897, Z -7.1667, A 0.000, B 0.000, C 0.000 }
gfCNCPoint5[11148] = {X 246.3936, Y 49.4000, Z -7.1667, A 0.000, B 0.000, C 0.000 }
gfCNCPoint5[11149] = {X 242.5312, Y 49.4000, Z -7.1667, A 0.000, B 0.000, C 0.000 }
gfCNCPoint5[11150] = {X 242.5312, Y 49.8800, Z -7.1667, A 0.000, B 0.000, C 0.000 }
gfCNCPoint5[11151] = {X 243.4812, Y 50.5824, Z -7.1667, A 0.000, B 0.000, C 0.000 }
gfCNCPoint5[11152] = {X 244.3384, Y 51.3953, Z -7.1667, A 0.000, B 0.000, C 0.000 }
gfCNCPoint5[11153] = {X 245.0903, Y 52.3066, Z -7.1667, A 0.000, B 0.000, C 0.000 }
gfCNCPoint5[11154] = {X 245.7256, Y 53.3027, Z -7.1667, A 0.000, B 0.000, C 0.000 }
gfCNCPoint5[11155] = {X 245.9754, Y 53.7841, Z -7.1667, A 0.000, B 0.000, C 0.000 }
gfCNCPoint5[11156] = {X 246.1978, Y 54.2787, Z -7.1667, A 0.000, B 0.000, C 0.000 }
gfCNCPoint5[11157] = {X 250.0866, Y 55.7952, Z -7.1667, A 0.000, B 0.000, C 0.000 }
gfCNCPoint5[11158] = {X 267.2821, Y 62.6204, Z -7.1667, A 0.000, B 0.000, C 0.000 }
gfCNCPoint5[11159] = {X 266.8842, Y 61.4458, Z -7.1667, A 0.000, B 0.000, C 0.000 }
gfCNCPoint5[11160] = {X 266.6398, Y 60.2300, Z -7.1667, A 0.000, B 0.000, C 0.000 }
gfCNCPoint5[11161] = {X 266.5529, Y 58.9930, Z -7.1667, A 0.000, B 0.000, C 0.000 }
gfCNCPoint5[11162] = {X 266.5527, Y 58.0000, Z -7.1667, A 0.000, B 0.000, C 0.000 }
gfCNCPoint5[11163] = {X 266.6262, Y 56.8093, Z -7.1667, A 0.000, B 0.000, C 0.000 }
gfCNCPoint5[11164] = {X 266.8456, Y 55.6367, Z -7.1667, A 0.000, B 0.000, C 0.000 }
gfCNCPoint5[11165] = {X 267.2076, Y 54.5000, Z -7.1667, A 0.000, B 0.000, C 0.000 }
gfCNCPoint5[11166] = {X 267.7067, Y 53.4164, Z -7.1667, A 0.000, B 0.000, C 0.000 }
gfCNCPoint5[11167] = {X 268.4728, Y 52.2132, Z -7.1667, A 0.000, B 0.000, C 0.000 }
gfCNCPoint5[11168] = {X 269.4075, Y 51.1357, Z -7.1667, A 0.000, B 0.000, C 0.000 }
gfCNCPoint5[11169] = {X 270.4903, Y 50.2072, Z -7.1667, A 0.000, B 0.000, C 0.000 }
gfCNCPoint5[11170] = {X 271.6979, Y 49.4479, Z -7.1667, A 0.000, B 0.000, C 0.000 }
gfCNCPoint5[11171] = {X 273.0039, Y 48.8744, Z -7.1667, A 0.000, B 0.000, C 0.000 }
gfCNCPoint5[11172] = {X 274.3800, Y 48.4989, Z -7.1667, A 0.000, B 0.000, C 0.000 }
gfCNCPoint5[11173] = {X 275.3020, Y 48.3648, Z -7.1667, A 0.000, B 0.000, C 0.000 }
gfCNCPoint5[11174] = {X 276.2327, Y 48.3200, Z -7.1667, A 0.000, B 0.000, C 0.000 }
gfCNCPoint5[11175] = {X 281.0411, Y 48.3200, Z -7.1667, A 0.000, B 0.000, C 0.000 }
gfCNCPoint5[11176] = {X 280.4347, Y 47.5134, Z -7.1667, A 0.000, B 0.000, C 0.000 }
gfCNCPoint5[11177] = {X 280.0072, Y 46.5992, Z -7.1667, A 0.000, B 0.000, C 0.000 }
gfCNCPoint5[11178] = {X 279.7768, Y 45.6167, Z -7.1667, A 0.000, B 0.000, C 0.000 }
gfCNCPoint5[11179] = {X 279.7488, Y 45.3288, Z -7.1667, A 0.000, B 0.000, C 0.000 }
gfCNCPoint5[11180] = {X 279.7378, Y 45.0398, Z -7.1667, A 0.000, B 0.000, C 0.000 }
gfCNCPoint5[11181] = {X 279.7377, Y 44.2050, Z -7.1667, A 0.000, B 0.000, C 0.000 }
gfCNCPoint5[11182] = {X 279.8414, Y 43.2211, Z -7.1667, A 0.000, B 0.000, C 0.000 }
gfCNCPoint5[11183] = {X 280.1396, Y 42.2777, Z -7.1667, A 0.000, B 0.000, C 0.000 }
gfCNCPoint5[11184] = {X 280.6205, Y 41.4131, Z -7.1667, A 0.000, B 0.000, C 0.000 }
gfCNCPoint5[11185] = {X 281.2644, Y 40.6619, Z -7.1667, A 0.000, B 0.000, C 0.000 }
gfCNCPoint5[11186] = {X 281.2643, Y 16.5233, Z -7.1667, A 0.000, B 0.000, C 0.000 }
gfCNCPoint5[11187] = {X 280.6235, Y 15.7818, Z -7.1667, A 0.000, B 0.000, C 0.000 }
gfCNCPoint5[11188] = {X 280.1438, Y 14.9272, Z -7.1667, A 0.000, B 0.000, C 0.000 }
gfCNCPoint5[11189] = {X 279.8446, Y 13.9940, Z -7.1667, A 0.000, B 0.000, C 0.000 }
gfCNCPoint5[11190] = {X 279.7378, Y 13.0198, Z -7.1667, A 0.000, B 0.000, C 0.000 }
gfCNCPoint5[11191] = {X 279.7377, Y 12.1868, Z -7.1667, A 0.000, B 0.000, C 0.000 }
gfCNCPoint5[11192] = {X 279.8242, Y 11.2717, Z -7.1667, A 0.000, B 0.000, C 0.000 }
gfCNCPoint5[11193] = {X 280.0809, Y 10.3890, Z -7.1667, A 0.000, B 0.000, C 0.000 }
gfCNCPoint5[11194] = {X 280.5256, Y 9.5280, Z -7.1667, A 0.000, B 0.000, C 0.000 }
gfCNCPoint5[11195] = {X 281.1317, Y 8.7718, Z -7.1667, A 0.000, B 0.000, C 0.000 }
gfCNCPoint5[11196] = {X 281.8753, Y 8.1503, Z -7.1667, A 0.000, B 0.000, C 0.000 }
gfCNCPoint5[11197] = {X 282.7270, Y 7.6879, Z -7.1667, A 0.000, B 0.000, C 0.000 }
gfCNCPoint5[11198] = {X 283.6533, Y 7.4030, Z -7.1667, A 0.000, B 0.000, C 0.000 }
gfCNCPoint5[11199] = {X 284.6177, Y 7.3068, Z -7.1667, A 0.000, B 0.000, C 0.000 }
gfCNCPoint5[11200] = {X 291.0611, Y 7.3068, Z -7.1667, A 0.000, B 0.000, C 0.000 }
gfCNCPoint5[11201] = {X 292.0255, Y 7.4030, Z -7.1667, A 0.000, B 0.000, C 0.000 }
gfCNCPoint5[11202] = {X 292.9518, Y 7.6879, Z -7.1667, A 0.000, B 0.000, C 0.000 }
gfCNCPoint5[11203] = {X 293.8035, Y 8.1503, Z -7.1667, A 0.000, B 0.000, C 0.000 }
gfCNCPoint5[11204] = {X 294.5471, Y 8.7718, Z -7.1667, A 0.000, B 0.000, C 0.000 }
gfCNCPoint5[11205] = {X 295.1532, Y 9.5280, Z -7.1667, A 0.000, B 0.000, C 0.000 }
gfCNCPoint5[11206] = {X 295.5979, Y 10.3890, Z -7.1667, A 0.000, B 0.000, C 0.000 }
gfCNCPoint5[11207] = {X 295.8044, Y 11.0396, Z -7.1667, A 0.000, B 0.000, C 0.000 }
gfCNCPoint5[11208] = {X 295.9181, Y 11.7127, Z -7.1667, A 0.000, B 0.000, C 0.000 }
gfCNCPoint5[11209] = {X 295.9354, Y 11.9495, Z -7.1667, A 0.000, B 0.000, C 0.000 }
gfCNCPoint5[11210] = {X 295.9411, Y 12.1868, Z -7.1667, A 0.000, B 0.000, C 0.000 }
gfCNCPoint5[11211] = {X 295.9409, Y 13.0237, Z -7.1667, A 0.000, B 0.000, C 0.000 }
gfCNCPoint5[11212] = {X 295.9342, Y 13.2382, Z -7.1667, A 0.000, B 0.000, C 0.000 }
gfCNCPoint5[11213] = {X 295.9180, Y 13.4521, Z -7.1667, A 0.000, B 0.000, C 0.000 }
gfCNCPoint5[11214] = {X 298.3067, Y 13.6853, Z -7.1667, A 0.000, B 0.000, C 0.000 }
gfCNCPoint5[11215] = {X 298.1362, Y 14.6932, Z -7.1667, A 0.000, B 0.000, C 0.000 }
gfCNCPoint5[11216] = {X 297.8262, Y 15.6674, Z -7.1667, A 0.000, B 0.000, C 0.000 }
gfCNCPoint5[11217] = {X 297.3827, Y 16.5885, Z -7.1667, A 0.000, B 0.000, C 0.000 }
gfCNCPoint5[11218] = {X 296.8147, Y 17.4384, Z -7.1667, A 0.000, B 0.000, C 0.000 }
gfCNCPoint5[11219] = {X 296.8149, Y 19.2365, Z -7.1667, A 0.000, B 0.000, C 0.000 }
gfCNCPoint5[11220] = {X 299.7984, Y 19.2365, Z -7.1667, A 0.000, B 0.000, C 0.000 }
gfCNCPoint5[11221] = {X 299.7985, Y 17.4381, Z -7.1667, A 0.000, B 0.000, C 0.000 }
gfCNCPoint5[11222] = {X 299.2305, Y 16.5882, Z -7.1667, A 0.000, B 0.000, C 0.000 }
gfCNCPoint5[11223] = {X 298.7871, Y 15.6672, Z -7.1667, A 0.000, B 0.000, C 0.000 }
gfCNCPoint5[11224] = {X 298.4772, Y 14.6931, Z -7.1667, A 0.000, B 0.000, C 0.000 }
gfCNCPoint5[11225] = {X 298.3067, Y 13.6853, Z -7.1667, A 0.000, B 0.000, C 0.000 }
gfCNCPoint5[11226] = {X 295.9180, Y 13.4521, Z -7.1667, A 0.000, B 0.000, C 0.000 }
gfCNCPoint5[11227] = {X 295.7561, Y 14.3092, Z -7.1667, A 0.000, B 0.000, C 0.000 }
gfCNCPoint5[11228] = {X 295.4441, Y 15.1237, Z -7.1667, A 0.000, B 0.000, C 0.000 }
gfCNCPoint5[11229] = {X 294.9921, Y 15.8697, Z -7.1667, A 0.000, B 0.000, C 0.000 }
gfCNCPoint5[11230] = {X 294.4145, Y 16.5233, Z -7.1667, A 0.000, B 0.000, C 0.000 }
gfCNCPoint5[11231] = {X 294.4153, Y 21.6365, Z -7.1667, A 0.000, B 0.000, C 0.000 }
gfCNCPoint5[11232] = {X 302.1983, Y 21.6365, Z -7.1667, A 0.000, B 0.000, C 0.000 }
gfCNCPoint5[11233] = {X 302.1985, Y 16.5230, Z -7.1667, A 0.000, B 0.000, C 0.000 }
gfCNCPoint5[11234] = {X 301.6211, Y 15.8694, Z -7.1667, A 0.000, B 0.000, C 0.000 }
gfCNCPoint5[11235] = {X 301.1692, Y 15.1235, Z -7.1667, A 0.000, B 0.000, C 0.000 }
gfCNCPoint5[11236] = {X 300.8573, Y 14.3091, Z -7.1667, A 0.000, B 0.000, C 0.000 }
gfCNCPoint5[11237] = {X 300.6953, Y 13.4521, Z -7.1667, A 0.000, B 0.000, C 0.000 }
gfCNCPoint5[11238] = {X 300.6791, Y 13.2371, Z -7.1667, A 0.000, B 0.000, C 0.000 }
gfCNCPoint5[11239] = {X 300.6724, Y 13.0215, Z -7.1667, A 0.000, B 0.000, C 0.000 }
gfCNCPoint5[11240] = {X 300.6723, Y 12.1868, Z -7.1667, A 0.000, B 0.000, C 0.000 }
gfCNCPoint5[11241] = {X 300.6780, Y 11.9495, Z -7.1667, A 0.000, B 0.000, C 0.000 }
gfCNCPoint5[11242] = {X 300.6953, Y 11.7127, Z -7.1667, A 0.000, B 0.000, C 0.000 }
gfCNCPoint5[11243] = {X 300.8090, Y 11.0396, Z -7.1667, A 0.000, B 0.000, C 0.000 }
gfCNCPoint5[11244] = {X 301.0155, Y 10.3890, Z -7.1667, A 0.000, B 0.000, C 0.000 }
gfCNCPoint5[11245] = {X 301.4602, Y 9.5280, Z -7.1667, A 0.000, B 0.000, C 0.000 }
gfCNCPoint5[11246] = {X 302.0663, Y 8.7718, Z -7.1667, A 0.000, B 0.000, C 0.000 }
gfCNCPoint5[11247] = {X 302.8099, Y 8.1503, Z -7.1667, A 0.000, B 0.000, C 0.000 }
gfCNCPoint5[11248] = {X 303.6616, Y 7.6879, Z -7.1667, A 0.000, B 0.000, C 0.000 }
gfCNCPoint5[11249] = {X 304.5879, Y 7.4030, Z -7.1667, A 0.000, B 0.000, C 0.000 }
gfCNCPoint5[11250] = {X 305.5523, Y 7.3068, Z -7.1667, A 0.000, B 0.000, C 0.000 }
gfCNCPoint5[11251] = {X 311.9957, Y 7.3068, Z -7.1667, A 0.000, B 0.000, C 0.000 }
gfCNCPoint5[11252] = {X 312.9478, Y 7.4006, Z -7.1667, A 0.000, B 0.000, C 0.000 }
gfCNCPoint5[11253] = {X 313.8632, Y 7.6783, Z -7.1667, A 0.000, B 0.000, C 0.000 }
gfCNCPoint5[11254] = {X 314.7069, Y 8.1292, Z -7.1667, A 0.000, B 0.000, C 0.000 }
gfCNCPoint5[11255] = {X 315.4464, Y 8.7361, Z -7.1667, A 0.000, B 0.000, C 0.000 }
gfCNCPoint5[11256] = {X 316.0533, Y 9.4756, Z -7.1667, A 0.000, B 0.000, C 0.000 }
gfCNCPoint5[11257] = {X 316.5043, Y 10.3193, Z -7.1667, A 0.000, B 0.000, C 0.000 }
gfCNCPoint5[11258] = {X 316.7820, Y 11.2348, Z -7.1667, A 0.000, B 0.000, C 0.000 }
gfCNCPoint5[11259] = {X 316.8757, Y 12.1868, Z -7.1667, A 0.000, B 0.000, C 0.000 }
gfCNCPoint5[11260] = {X 316.8755, Y 13.0237, Z -7.1667, A 0.000, B 0.000, C 0.000 }
gfCNCPoint5[11261] = {X 316.7682, Y 13.9967, Z -7.1667, A 0.000, B 0.000, C 0.000 }
gfCNCPoint5[11262] = {X 316.4689, Y 14.9287, Z -7.1667, A 0.000, B 0.000, C 0.000 }
gfCNCPoint5[11263] = {X 315.9895, Y 15.7823, Z -7.1667, A 0.000, B 0.000, C 0.000 }
gfCNCPoint5[11264] = {X 315.3495, Y 16.5229, Z -7.1667, A 0.000, B 0.000, C 0.000 }
gfCNCPoint5[11265] = {X 315.3490, Y 40.6634, Z -7.1667, A 0.000, B 0.000, C 0.000 }
gfCNCPoint5[11266] = {X 315.9897, Y 41.4048, Z -7.1667, A 0.000, B 0.000, C 0.000 }
gfCNCPoint5[11267] = {X 316.4694, Y 42.2593, Z -7.1667, A 0.000, B 0.000, C 0.000 }
gfCNCPoint5[11268] = {X 316.7687, Y 43.1924, Z -7.1667, A 0.000, B 0.000, C 0.000 }
gfCNCPoint5[11269] = {X 316.8755, Y 44.1664, Z -7.1667, A 0.000, B 0.000, C 0.000 }
gfCNCPoint5[11270] = {X 316.8757, Y 45.0000, Z -7.1667, A 0.000, B 0.000, C 0.000 }
gfCNCPoint5[11271] = {X 316.8749, Y 45.0899, Z -7.1667, A 0.000, B 0.000, C 0.000 }
gfCNCPoint5[11272] = {X 316.8724, Y 45.1799, Z -7.1667, A 0.000, B 0.000, C 0.000 }
gfCNCPoint5[11273] = {X 316.8594, Y 45.3987, Z -7.1667, A 0.000, B 0.000, C 0.000 }
gfCNCPoint5[11274] = {X 316.8366, Y 45.6167, Z -7.1667, A 0.000, B 0.000, C 0.000 }
gfCNCPoint5[11275] = {X 316.6062, Y 46.5992, Z -7.1667, A 0.000, B 0.000, C 0.000 }
gfCNCPoint5[11276] = {X 316.1787, Y 47.5134, Z -7.1667, A 0.000, B 0.000, C 0.000 }
gfCNCPoint5[11277] = {X 315.5723, Y 48.3200, Z -7.1667, A 0.000, B 0.000, C 0.000 }
gfCNCPoint5[11278] = {X 315.2205, Y 47.9934, Z -7.1667, A 0.000, B 0.000, C 0.000 }
gfCNCPoint5[11279] = {X 314.5413, Y 48.5889, Z -7.1667, A 0.000, B 0.000, C 0.000 }
gfCNCPoint5[11280] = {X 313.7548, Y 49.0331, Z -7.1667, A 0.000, B 0.000, C 0.000 }
gfCNCPoint5[11281] = {X 312.8942, Y 49.3073, Z -7.1667, A 0.000, B 0.000, C 0.000 }
gfCNCPoint5[11282] = {X 311.9957, Y 49.4000, Z -7.1667, A 0.000, B 0.000, C 0.000 }
gfCNCPoint5[11283] = {X 305.5523, Y 49.4000, Z -7.1667, A 0.000, B 0.000, C 0.000 }
gfCNCPoint5[11284] = {X 304.5732, Y 49.2897, Z -7.1667, A 0.000, B 0.000, C 0.000 }
gfCNCPoint5[11285] = {X 303.6432, Y 48.9643, Z -7.1667, A 0.000, B 0.000, C 0.000 }
gfCNCPoint5[11286] = {X 302.8089, Y 48.4400, Z -7.1667, A 0.000, B 0.000, C 0.000 }
gfCNCPoint5[11287] = {X 302.1122, Y 47.7433, Z -7.1667, A 0.000, B 0.000, C 0.000 }
gfCNCPoint5[11288] = {X 301.5880, Y 46.9091, Z -7.1667, A 0.000, B 0.000, C 0.000 }
gfCNCPoint5[11289] = {X 301.2626, Y 45.9791, Z -7.1667, A 0.000, B 0.000, C 0.000 }
gfCNCPoint5[11290] = {X 301.1523, Y 45.0000, Z -7.1667, A 0.000, B 0.000, C 0.000 }
gfCNCPoint5[11291] = {X 301.1524, Y 44.1995, Z -7.1667, A 0.000, B 0.000, C 0.000 }
gfCNCPoint5[11292] = {X 301.2695, Y 43.2560, Z -7.1667, A 0.000, B 0.000, C 0.000 }
gfCNCPoint5[11293] = {X 301.5722, Y 42.3548, Z -7.1667, A 0.000, B 0.000, C 0.000 }
gfCNCPoint5[11294] = {X 302.0483, Y 41.5318, Z -7.1667, A 0.000, B 0.000, C 0.000 }
gfCNCPoint5[11295] = {X 302.6787, Y 40.8201, Z -7.1667, A 0.000, B 0.000, C 0.000 }
gfCNCPoint5[11296] = {X 302.6787, Y 34.1143, Z -7.1667, A 0.000, B 0.000, C 0.000 }
gfCNCPoint5[11297] = {X 293.9352, Y 34.1143, Z -7.1667, A 0.000, B 0.000, C 0.000 }
gfCNCPoint5[11298] = {X 293.9346, Y 40.8655, Z -7.1667, A 0.000, B 0.000, C 0.000 }
gfCNCPoint5[11299] = {X 294.5746, Y 41.5605, Z -7.1667, A 0.000, B 0.000, C 0.000 }
gfCNCPoint5[11300] = {X 295.0553, Y 42.3740, Z -7.1667, A 0.000, B 0.000, C 0.000 }
gfCNCPoint5[11301] = {X 295.3552, Y 43.2700, Z -7.1667, A 0.000, B 0.000, C 0.000 }
gfCNCPoint5[11302] = {X 295.4611, Y 44.2089, Z -7.1667, A 0.000, B 0.000, C 0.000 }
gfCNCPoint5[11303] = {X 295.4611, Y 45.0000, Z -7.1667, A 0.000, B 0.000, C 0.000 }
gfCNCPoint5[11304] = {X 295.3508, Y 45.9791, Z -7.1667, A 0.000, B 0.000, C 0.000 }
gfCNCPoint5[11305] = {X 295.0254, Y 46.9091, Z -7.1667, A 0.000, B 0.000, C 0.000 }
gfCNCPoint5[11306] = {X 294.5012, Y 47.7434, Z -7.1667, A 0.000, B 0.000, C 0.000 }
gfCNCPoint5[11307] = {X 293.8045, Y 48.4401, Z -7.1667, A 0.000, B 0.000, C 0.000 }
gfCNCPoint5[11308] = {X 292.9702, Y 48.9643, Z -7.1667, A 0.000, B 0.000, C 0.000 }
gfCNCPoint5[11309] = {X 292.0402, Y 49.2897, Z -7.1667, A 0.000, B 0.000, C 0.000 }
gfCNCPoint5[11310] = {X 291.0611, Y 49.4000, Z -7.1667, A 0.000, B 0.000, C 0.000 }
gfCNCPoint5[11311] = {X 284.6177, Y 49.4000, Z -7.1667, A 0.000, B 0.000, C 0.000 }
gfCNCPoint5[11312] = {X 283.6386, Y 49.2897, Z -7.1667, A 0.000, B 0.000, C 0.000 }
gfCNCPoint5[11313] = {X 282.7086, Y 48.9643, Z -7.1667, A 0.000, B 0.000, C 0.000 }
gfCNCPoint5[11314] = {X 281.8743, Y 48.4401, Z -7.1667, A 0.000, B 0.000, C 0.000 }
gfCNCPoint5[11315] = {X 281.1776, Y 47.7433, Z -7.1667, A 0.000, B 0.000, C 0.000 }
gfCNCPoint5[11316] = {X 280.6534, Y 46.9091, Z -7.1667, A 0.000, B 0.000, C 0.000 }
gfCNCPoint5[11317] = {X 280.3280, Y 45.9791, Z -7.1667, A 0.000, B 0.000, C 0.000 }
gfCNCPoint5[11318] = {X 280.2177, Y 45.0000, Z -7.1667, A 0.000, B 0.000, C 0.000 }
gfCNCPoint5[11319] = {X 280.2177, Y 44.2071, Z -7.1667, A 0.000, B 0.000, C 0.000 }
gfCNCPoint5[11320] = {X 280.3218, Y 43.2699, Z -7.1667, A 0.000, B 0.000, C 0.000 }
gfCNCPoint5[11321] = {X 280.6213, Y 42.3757, Z -7.1667, A 0.000, B 0.000, C 0.000 }
gfCNCPoint5[11322] = {X 281.1028, Y 41.5648, Z -7.1667, A 0.000, B 0.000, C 0.000 }
gfCNCPoint5[11323] = {X 281.7444, Y 40.8738, Z -7.1667, A 0.000, B 0.000, C 0.000 }
gfCNCPoint5[11324] = {X 281.7443, Y 16.3102, Z -7.1667, A 0.000, B 0.000, C 0.000 }
gfCNCPoint5[11325] = {X 281.1000, Y 15.6212, Z -7.1667, A 0.000, B 0.000, C 0.000 }
gfCNCPoint5[11326] = {X 280.6175, Y 14.8106, Z -7.1667, A 0.000, B 0.000, C 0.000 }
gfCNCPoint5[11327] = {X 280.3188, Y 13.9159, Z -7.1667, A 0.000, B 0.000, C 0.000 }
gfCNCPoint5[11328] = {X 280.2177, Y 12.9780, Z -7.1667, A 0.000, B 0.000, C 0.000 }
gfCNCPoint5[11329] = {X 280.2177, Y 12.1868, Z -7.1667, A 0.000, B 0.000, C 0.000 }
gfCNCPoint5[11330] = {X 280.3280, Y 11.2077, Z -7.1667, A 0.000, B 0.000, C 0.000 }
gfCNCPoint5[11331] = {X 280.6534, Y 10.2777, Z -7.1667, A 0.000, B 0.000, C 0.000 }
gfCNCPoint5[11332] = {X 281.1776, Y 9.4435, Z -7.1667, A 0.000, B 0.000, C 0.000 }
gfCNCPoint5[11333] = {X 281.8743, Y 8.7468, Z -7.1667, A 0.000, B 0.000, C 0.000 }
gfCNCPoint5[11334] = {X 282.7086, Y 8.2226, Z -7.1667, A 0.000, B 0.000, C 0.000 }
gfCNCPoint5[11335] = {X 283.6386, Y 7.8971, Z -7.1667, A 0.000, B 0.000, C 0.000 }
gfCNCPoint5[11336] = {X 284.6177, Y 7.7868, Z -7.1667, A 0.000, B 0.000, C 0.000 }
gfCNCPoint5[11337] = {X 291.0611, Y 7.7868, Z -7.1667, A 0.000, B 0.000, C 0.000 }
gfCNCPoint5[11338] = {X 292.0402, Y 7.8971, Z -7.1667, A 0.000, B 0.000, C 0.000 }
gfCNCPoint5[11339] = {X 292.9702, Y 8.2226, Z -7.1667, A 0.000, B 0.000, C 0.000 }
gfCNCPoint5[11340] = {X 293.8045, Y 8.7468, Z -7.1667, A 0.000, B 0.000, C 0.000 }
gfCNCPoint5[11341] = {X 294.5012, Y 9.4435, Z -7.1667, A 0.000, B 0.000, C 0.000 }
gfCNCPoint5[11342] = {X 295.0254, Y 10.2777, Z -7.1667, A 0.000, B 0.000, C 0.000 }
gfCNCPoint5[11343] = {X 295.3508, Y 11.2077, Z -7.1667, A 0.000, B 0.000, C 0.000 }
gfCNCPoint5[11344] = {X 295.4611, Y 12.1868, Z -7.1667, A 0.000, B 0.000, C 0.000 }
gfCNCPoint5[11345] = {X 295.4609, Y 13.0233, Z -7.1667, A 0.000, B 0.000, C 0.000 }
gfCNCPoint5[11346] = {X 295.3526, Y 13.9491, Z -7.1667, A 0.000, B 0.000, C 0.000 }
gfCNCPoint5[11347] = {X 295.0518, Y 14.8312, Z -7.1667, A 0.000, B 0.000, C 0.000 }
gfCNCPoint5[11348] = {X 294.5719, Y 15.6303, Z -7.1667, A 0.000, B 0.000, C 0.000 }
gfCNCPoint5[11349] = {X 293.9345, Y 16.3103, Z -7.1667, A 0.000, B 0.000, C 0.000 }
gfCNCPoint5[11350] = {X 293.9354, Y 22.1165, Z -7.1667, A 0.000, B 0.000, C 0.000 }
gfCNCPoint5[11351] = {X 302.6783, Y 22.1165, Z -7.1667, A 0.000, B 0.000, C 0.000 }
gfCNCPoint5[11352] = {X 302.6785, Y 16.3099, Z -7.1667, A 0.000, B 0.000, C 0.000 }
gfCNCPoint5[11353] = {X 302.0344, Y 15.6209, Z -7.1667, A 0.000, B 0.000, C 0.000 }
gfCNCPoint5[11354] = {X 301.5520, Y 14.8104, Z -7.1667, A 0.000, B 0.000, C 0.000 }
gfCNCPoint5[11355] = {X 301.2533, Y 13.9157, Z -7.1667, A 0.000, B 0.000, C 0.000 }
gfCNCPoint5[11356] = {X 301.1523, Y 12.9780, Z -7.1667, A 0.000, B 0.000, C 0.000 }
gfCNCPoint5[11357] = {X 301.1523, Y 12.1868, Z -7.1667, A 0.000, B 0.000, C 0.000 }
gfCNCPoint5[11358] = {X 301.2626, Y 11.2077, Z -7.1667, A 0.000, B 0.000, C 0.000 }
gfCNCPoint5[11359] = {X 301.5880, Y 10.2777, Z -7.1667, A 0.000, B 0.000, C 0.000 }
gfCNCPoint5[11360] = {X 302.1122, Y 9.4435, Z -7.1667, A 0.000, B 0.000, C 0.000 }
gfCNCPoint5[11361] = {X 302.8089, Y 8.7468, Z -7.1667, A 0.000, B 0.000, C 0.000 }
gfCNCPoint5[11362] = {X 303.6432, Y 8.2226, Z -7.1667, A 0.000, B 0.000, C 0.000 }
gfCNCPoint5[11363] = {X 304.5732, Y 7.8971, Z -7.1667, A 0.000, B 0.000, C 0.000 }
gfCNCPoint5[11364] = {X 305.5523, Y 7.7868, Z -7.1667, A 0.000, B 0.000, C 0.000 }
gfCNCPoint5[11365] = {X 311.9957, Y 7.7868, Z -7.1667, A 0.000, B 0.000, C 0.000 }
gfCNCPoint5[11366] = {X 312.9748, Y 7.8971, Z -7.1667, A 0.000, B 0.000, C 0.000 }
gfCNCPoint5[11367] = {X 313.9048, Y 8.2226, Z -7.1667, A 0.000, B 0.000, C 0.000 }
gfCNCPoint5[11368] = {X 314.7391, Y 8.7468, Z -7.1667, A 0.000, B 0.000, C 0.000 }
gfCNCPoint5[11369] = {X 315.4358, Y 9.4435, Z -7.1667, A 0.000, B 0.000, C 0.000 }
gfCNCPoint5[11370] = {X 315.9600, Y 10.2777, Z -7.1667, A 0.000, B 0.000, C 0.000 }
gfCNCPoint5[11371] = {X 316.2854, Y 11.2077, Z -7.1667, A 0.000, B 0.000, C 0.000 }
gfCNCPoint5[11372] = {X 316.3957, Y 12.1868, Z -7.1667, A 0.000, B 0.000, C 0.000 }
gfCNCPoint5[11373] = {X 316.3955, Y 13.0233, Z -7.1667, A 0.000, B 0.000, C 0.000 }
gfCNCPoint5[11374] = {X 316.2873, Y 13.9489, Z -7.1667, A 0.000, B 0.000, C 0.000 }
gfCNCPoint5[11375] = {X 315.9865, Y 14.8310, Z -7.1667, A 0.000, B 0.000, C 0.000 }
gfCNCPoint5[11376] = {X 315.5068, Y 15.6299, Z -7.1667, A 0.000, B 0.000, C 0.000 }
gfCNCPoint5[11377] = {X 314.8695, Y 16.3099, Z -7.1667, A 0.000, B 0.000, C 0.000 }
gfCNCPoint5[11378] = {X 314.8690, Y 40.8765, Z -7.1667, A 0.000, B 0.000, C 0.000 }
gfCNCPoint5[11379] = {X 315.5133, Y 41.5656, Z -7.1667, A 0.000, B 0.000, C 0.000 }
gfCNCPoint5[11380] = {X 315.9959, Y 42.3761, Z -7.1667, A 0.000, B 0.000, C 0.000 }
gfCNCPoint5[11381] = {X 316.2946, Y 43.2709, Z -7.1667, A 0.000, B 0.000, C 0.000 }
gfCNCPoint5[11382] = {X 316.3957, Y 44.2089, Z -7.1667, A 0.000, B 0.000, C 0.000 }
gfCNCPoint5[11383] = {X 316.3957, Y 45.0000, Z -7.1667, A 0.000, B 0.000, C 0.000 }
gfCNCPoint5[11384] = {X 316.3190, Y 45.8182, Z -7.1667, A 0.000, B 0.000, C 0.000 }
gfCNCPoint5[11385] = {X 316.0914, Y 46.6079, Z -7.1667, A 0.000, B 0.000, C 0.000 }
gfCNCPoint5[11386] = {X 315.7209, Y 47.3415, Z -7.1667, A 0.000, B 0.000, C 0.000 }
gfCNCPoint5[11387] = {X 315.2205, Y 47.9934, Z -7.1667, A 0.000, B 0.000, C 0.000 }
gfCNCPoint5[11388] = {X 315.5723, Y 48.3200, Z -7.1667, A 0.000, B 0.000, C 0.000 }
gfCNCPoint5[11389] = {X 324.3107, Y 48.3200, Z -7.1667, A 0.000, B 0.000, C 0.000 }
gfCNCPoint5[11390] = {X 325.5555, Y 48.4004, Z -7.1667, A 0.000, B 0.000, C 0.000 }
gfCNCPoint5[11391] = {X 326.7797, Y 48.6402, Z -7.1667, A 0.000, B 0.000, C 0.000 }
gfCNCPoint5[11392] = {X 325.5882, Y 48.0963, Z -7.1667, A 0.000, B 0.000, C 0.000 }
gfCNCPoint5[11393] = {X 324.4810, Y 47.3966, Z -7.1667, A 0.000, B 0.000, C 0.000 }
gfCNCPoint5[11394] = {X 323.4784, Y 46.5538, Z -7.1667, A 0.000, B 0.000, C 0.000 }
gfCNCPoint5[11395] = {X 322.8382, Y 45.9295, Z -7.1667, A 0.000, B 0.000, C 0.000 }
gfCNCPoint5[11396] = {X 322.2180, Y 45.2650, Z -7.1667, A 0.000, B 0.000, C 0.000 }
gfCNCPoint5[11397] = {X 321.6628, Y 44.5452, Z -7.1667, A 0.000, B 0.000, C 0.000 }
gfCNCPoint5[11398] = {X 323.6300, Y 43.1703, Z -7.1667, A 0.000, B 0.000, C 0.000 }
gfCNCPoint5[11399] = {X 323.0063, Y 42.0918, Z -7.1667, A 0.000, B 0.000, C 0.000 }
gfCNCPoint5[11400] = {X 322.5757, Y 40.9227, Z -7.1667, A 0.000, B 0.000, C 0.000 }
gfCNCPoint5[11401] = {X 322.3506, Y 39.6973, Z -7.1667, A 0.000, B 0.000, C 0.000 }
gfCNCPoint5[11402] = {X 322.3379, Y 38.4514, Z -7.1667, A 0.000, B 0.000, C 0.000 }
gfCNCPoint5[11403] = {X 322.5377, Y 37.2217, Z -7.1667, A 0.000, B 0.000, C 0.000 }
gfCNCPoint5[11404] = {X 322.9443, Y 36.0440, Z -7.1667, A 0.000, B 0.000, C 0.000 }
gfCNCPoint5[11405] = {X 323.5458, Y 34.9529, Z -7.1667, A 0.000, B 0.000, C 0.000 }
gfCNCPoint5[11406] = {X 327.7841, Y 28.6158, Z -7.1667, A 0.000, B 0.000, C 0.000 }
gfCNCPoint5[11407] = {X 328.5200, Y 27.6906, Z -7.1667, A 0.000, B 0.000, C 0.000 }
gfCNCPoint5[11408] = {X 329.3960, Y 26.8968, Z -7.1667, A 0.000, B 0.000, C 0.000 }
gfCNCPoint5[11409] = {X 330.3889, Y 26.2552, Z -7.1667, A 0.000, B 0.000, C 0.000 }
gfCNCPoint5[11410] = {X 331.5063, Y 25.7713, Z -7.1667, A 0.000, B 0.000, C 0.000 }
gfCNCPoint5[11411] = {X 332.6887, Y 25.4804, Z -7.1667, A 0.000, B 0.000, C 0.000 }
gfCNCPoint5[11412] = {X 333.9031, Y 25.3907, Z -7.1667, A 0.000, B 0.000, C 0.000 }
gfCNCPoint5[11413] = {X 335.1154, Y 25.5046, Z -7.1667, A 0.000, B 0.000, C 0.000 }
gfCNCPoint5[11414] = {X 336.2918, Y 25.8191, Z -7.1667, A 0.000, B 0.000, C 0.000 }
gfCNCPoint5[11415] = {X 337.3993, Y 26.3252, Z -7.1667, A 0.000, B 0.000, C 0.000 }
gfCNCPoint5[11416] = {X 338.1754, Y 26.8291, Z -7.1667, A 0.000, B 0.000, C 0.000 }
gfCNCPoint5[11417] = {X 338.8812, Y 27.4274, Z -7.1667, A 0.000, B 0.000, C 0.000 }
gfCNCPoint5[11418] = {X 339.5028, Y 28.0267, Z -7.1667, A 0.000, B 0.000, C 0.000 }
gfCNCPoint5[11419] = {X 340.3318, Y 28.9981, Z -7.1667, A 0.000, B 0.000, C 0.000 }
gfCNCPoint5[11420] = {X 340.9782, Y 30.0994, Z -7.1667, A 0.000, B 0.000, C 0.000 }
gfCNCPoint5[11421] = {X 341.4222, Y 31.2968, Z -7.1667, A 0.000, B 0.000, C 0.000 }
gfCNCPoint5[11422] = {X 341.6502, Y 32.5533, Z -7.1667, A 0.000, B 0.000, C 0.000 }
gfCNCPoint5[11423] = {X 342.6387, Y 33.2802, Z -7.1667, A 0.000, B 0.000, C 0.000 }
gfCNCPoint5[11424] = {X 343.7299, Y 33.8415, Z -7.1667, A 0.000, B 0.000, C 0.000 }
gfCNCPoint5[11425] = {X 344.8961, Y 34.2230, Z -7.1667, A 0.000, B 0.000, C 0.000 }
gfCNCPoint5[11426] = {X 346.1080, Y 34.4149, Z -7.1667, A 0.000, B 0.000, C 0.000 }
gfCNCPoint5[11427] = {X 347.3351, Y 34.4126, Z -7.1667, A 0.000, B 0.000, C 0.000 }
gfCNCPoint5[11428] = {X 348.3042, Y 34.2870, Z -7.1667, A 0.000, B 0.000, C 0.000 }
gfCNCPoint5[11429] = {X 349.2395, Y 34.0039, Z -7.1667, A 0.000, B 0.000, C 0.000 }
gfCNCPoint5[11430] = {X 350.1157, Y 33.5712, Z -7.1667, A 0.000, B 0.000, C 0.000 }
gfCNCPoint5[11431] = {X 350.9091, Y 33.0006, Z -7.1667, A 0.000, B 0.000, C 0.000 }
gfCNCPoint5[11432] = {X 351.7850, Y 32.1496, Z -7.1667, A 0.000, B 0.000, C 0.000 }
gfCNCPoint5[11433] = {X 352.5432, Y 31.1922, Z -7.1667, A 0.000, B 0.000, C 0.000 }
gfCNCPoint5[11434] = {X 353.1709, Y 30.1446, Z -7.1667, A 0.000, B 0.000, C 0.000 }
gfCNCPoint5[11435] = {X 353.6575, Y 29.0245, Z -7.1667, A 0.000, B 0.000, C 0.000 }
gfCNCPoint5[11436] = {X 353.9948, Y 27.8508, Z -7.1667, A 0.000, B 0.000, C 0.000 }
gfCNCPoint5[11437] = {X 354.2223, Y 26.4400, Z -7.1667, A 0.000, B 0.000, C 0.000 }
gfCNCPoint5[11438] = {X 354.3143, Y 25.0140, Z -7.1667, A 0.000, B 0.000, C 0.000 }
gfCNCPoint5[11439] = {X 354.2701, Y 23.5857, Z -7.1667, A 0.000, B 0.000, C 0.000 }
gfCNCPoint5[11440] = {X 354.0900, Y 22.1681, Z -7.1667, A 0.000, B 0.000, C 0.000 }
gfCNCPoint5[11441] = {X 353.8252, Y 21.0253, Z -7.1667, A 0.000, B 0.000, C 0.000 }
gfCNCPoint5[11442] = {X 353.4121, Y 19.9274, Z -7.1667, A 0.000, B 0.000, C 0.000 }
gfCNCPoint5[11443] = {X 352.8577, Y 18.8935, Z -7.1667, A 0.000, B 0.000, C 0.000 }
gfCNCPoint5[11444] = {X 352.1718, Y 17.9418, Z -7.1667, A 0.000, B 0.000, C 0.000 }
gfCNCPoint5[11445] = {X 351.4219, Y 17.1687, Z -7.1667, A 0.000, B 0.000, C 0.000 }
gfCNCPoint5[11446] = {X 350.5492, Y 16.5373, Z -7.1667, A 0.000, B 0.000, C 0.000 }
gfCNCPoint5[11447] = {X 349.5804, Y 16.0668, Z -7.1667, A 0.000, B 0.000, C 0.000 }
gfCNCPoint5[11448] = {X 348.5446, Y 15.7714, Z -7.1667, A 0.000, B 0.000, C 0.000 }
gfCNCPoint5[11449] = {X 347.1584, Y 15.5993, Z -7.1667, A 0.000, B 0.000, C 0.000 }
gfCNCPoint5[11450] = {X 345.7616, Y 15.6145, Z -7.1667, A 0.000, B 0.000, C 0.000 }
gfCNCPoint5[11451] = {X 344.3795, Y 15.8167, Z -7.1667, A 0.000, B 0.000, C 0.000 }
gfCNCPoint5[11452] = {X 343.0369, Y 16.2022, Z -7.1667, A 0.000, B 0.000, C 0.000 }
gfCNCPoint5[11453] = {X 341.7581, Y 16.7642, Z -7.1667, A 0.000, B 0.000, C 0.000 }
gfCNCPoint5[11454] = {X 341.4305, Y 17.8588, Z -7.1667, A 0.000, B 0.000, C 0.000 }
gfCNCPoint5[11455] = {X 340.9357, Y 18.8887, Z -7.1667, A 0.000, B 0.000, C 0.000 }
gfCNCPoint5[11456] = {X 340.2859, Y 19.8284, Z -7.1667, A 0.000, B 0.000, C 0.000 }
gfCNCPoint5[11457] = {X 345.8684, Y 24.3755, Z -7.1667, A 0.000, B 0.000, C 0.000 }
gfCNCPoint5[11458] = {X 346.4661, Y 25.2108, Z -7.1667, A 0.000, B 0.000, C 0.000 }
gfCNCPoint5[11459] = {X 347.0031, Y 26.0864, Z -7.1667, A 0.000, B 0.000, C 0.000 }
gfCNCPoint5[11460] = {X 347.1052, Y 25.1807, Z -7.1667, A 0.000, B 0.000, C 0.000 }
gfCNCPoint5[11461] = {X 347.1008, Y 24.2693, Z -7.1667, A 0.000, B 0.000, C 0.000 }
gfCNCPoint5[11462] = {X 346.9899, Y 23.3647, Z -7.1667, A 0.000, B 0.000, C 0.000 }
gfCNCPoint5[11463] = {X 346.9486, Y 23.1617, Z -7.1667, A 0.000, B 0.000, C 0.000 }
gfCNCPoint5[11464] = {X 346.8826, Y 22.9654, Z -7.1667, A 0.000, B 0.000, C 0.000 }
gfCNCPoint5[11465] = {X 346.3966, Y 23.6857, Z -7.1667, A 0.000, B 0.000, C 0.000 }
gfCNCPoint5[11466] = {X 345.8684, Y 24.3755, Z -7.1667, A 0.000, B 0.000, C 0.000 }
gfCNCPoint5[11467] = {X 344.0076, Y 22.8598, Z -7.1667, A 0.000, B 0.000, C 0.000 }
gfCNCPoint5[11468] = {X 343.3277, Y 23.6257, Z -7.1667, A 0.000, B 0.000, C 0.000 }
gfCNCPoint5[11469] = {X 342.5854, Y 24.3313, Z -7.1667, A 0.000, B 0.000, C 0.000 }
gfCNCPoint5[11470] = {X 343.4621, Y 25.2276, Z -7.1667, A 0.000, B 0.000, C 0.000 }
gfCNCPoint5[11471] = {X 344.2411, Y 26.2100, Z -7.1667, A 0.000, B 0.000, C 0.000 }
gfCNCPoint5[11472] = {X 344.9141, Y 27.2678, Z -7.1667, A 0.000, B 0.000, C 0.000 }
gfCNCPoint5[11473] = {X 345.4657, Y 28.3713, Z -7.1667, A 0.000, B 0.000, C 0.000 }
gfCNCPoint5[11474] = {X 345.9020, Y 29.5253, Z -7.1667, A 0.000, B 0.000, C 0.000 }
gfCNCPoint5[11475] = {X 346.4628, Y 29.6285, Z -7.1667, A 0.000, B 0.000, C 0.000 }
gfCNCPoint5[11476] = {X 347.0330, Y 29.6209, Z -7.1667, A 0.000, B 0.000, C 0.000 }
gfCNCPoint5[11477] = {X 347.4389, Y 29.5548, Z -7.1667, A 0.000, B 0.000, C 0.000 }
gfCNCPoint5[11478] = {X 347.7946, Y 29.3482, Z -7.1667, A 0.000, B 0.000, C 0.000 }
gfCNCPoint5[11479] = {X 348.4744, Y 28.6288, Z -7.1667, A 0.000, B 0.000, C 0.000 }
gfCNCPoint5[11480] = {X 348.9846, Y 27.7807, Z -7.1667, A 0.000, B 0.000, C 0.000 }
gfCNCPoint5[11481] = {X 349.3018, Y 26.8432, Z -7.1667, A 0.000, B 0.000, C 0.000 }
gfCNCPoint5[11482] = {X 349.3365, Y 26.6690, Z -7.1667, A 0.000, B 0.000, C 0.000 }
gfCNCPoint5[11483] = {X 349.3682, Y 26.4943, Z -7.1667, A 0.000, B 0.000, C 0.000 }
gfCNCPoint5[11484] = {X 349.5011, Y 25.3212, Z -7.1667, A 0.000, B 0.000, C 0.000 }
gfCNCPoint5[11485] = {X 349.4974, Y 24.1407, Z -7.1667, A 0.000, B 0.000, C 0.000 }
gfCNCPoint5[11486] = {X 349.3571, Y 22.9685, Z -7.1667, A 0.000, B 0.000, C 0.000 }
gfCNCPoint5[11487] = {X 349.1794, Y 22.2565, Z -7.1667, A 0.000, B 0.000, C 0.000 }
gfCNCPoint5[11488] = {X 348.8769, Y 21.5880, Z -7.1667, A 0.000, B 0.000, C 0.000 }
gfCNCPoint5[11489] = {X 348.4594, Y 20.9845, Z -7.1667, A 0.000, B 0.000, C 0.000 }
gfCNCPoint5[11490] = {X 348.0918, Y 20.6606, Z -7.1667, A 0.000, B 0.000, C 0.000 }
gfCNCPoint5[11491] = {X 347.6347, Y 20.4843, Z -7.1667, A 0.000, B 0.000, C 0.000 }
gfCNCPoint5[11492] = {X 346.5775, Y 20.3828, Z -7.1667, A 0.000, B 0.000, C 0.000 }
gfCNCPoint5[11493] = {X 345.5201, Y 20.4826, Z -7.1667, A 0.000, B 0.000, C 0.000 }
gfCNCPoint5[11494] = {X 344.8334, Y 21.7155, Z -7.1667, A 0.000, B 0.000, C 0.000 }
gfCNCPoint5[11495] = {X 344.0076, Y 22.8598, Z -7.1667, A 0.000, B 0.000, C 0.000 }
gfCNCPoint5[11496] = {X 342.1467, Y 21.3441, Z -7.1667, A 0.000, B 0.000, C 0.000 }
gfCNCPoint5[11497] = {X 341.6020, Y 21.9578, Z -7.1667, A 0.000, B 0.000, C 0.000 }
gfCNCPoint5[11498] = {X 341.0072, Y 22.5232, Z -7.1667, A 0.000, B 0.000, C 0.000 }
gfCNCPoint5[11499] = {X 340.7216, Y 22.7630, Z -7.1667, A 0.000, B 0.000, C 0.000 }
gfCNCPoint5[11500] = {X 340.4270, Y 22.9916, Z -7.1667, A 0.000, B 0.000, C 0.000 }
gfCNCPoint5[11501] = {X 339.6615, Y 23.5549, Z -7.1667, A 0.000, B 0.000, C 0.000 }
gfCNCPoint5[11502] = {X 339.1299, Y 23.9121, Z -7.1667, A 0.000, B 0.000, C 0.000 }
gfCNCPoint5[11503] = {X 338.5759, Y 24.2333, Z -7.1667, A 0.000, B 0.000, C 0.000 }
gfCNCPoint5[11504] = {X 339.6078, Y 24.9034, Z -7.1667, A 0.000, B 0.000, C 0.000 }
gfCNCPoint5[11505] = {X 340.5463, Y 25.6990, Z -7.1667, A 0.000, B 0.000, C 0.000 }
gfCNCPoint5[11506] = {X 341.1848, Y 26.3147, Z -7.1667, A 0.000, B 0.000, C 0.000 }
gfCNCPoint5[11507] = {X 342.1205, Y 27.3795, Z -7.1667, A 0.000, B 0.000, C 0.000 }
gfCNCPoint5[11508] = {X 342.8906, Y 28.5695, Z -7.1667, A 0.000, B 0.000, C 0.000 }
gfCNCPoint5[11509] = {X 343.4787, Y 29.8592, Z -7.1667, A 0.000, B 0.000, C 0.000 }
gfCNCPoint5[11510] = {X 343.8722, Y 31.2210, Z -7.1667, A 0.000, B 0.000, C 0.000 }
gfCNCPoint5[11511] = {X 344.6396, Y 31.6206, Z -7.1667, A 0.000, B 0.000, C 0.000 }
gfCNCPoint5[11512] = {X 345.4616, Y 31.8906, Z -7.1667, A 0.000, B 0.000, C 0.000 }
gfCNCPoint5[11513] = {X 346.3165, Y 32.0240, Z -7.1667, A 0.000, B 0.000, C 0.000 }
gfCNCPoint5[11514] = {X 347.1817, Y 32.0172, Z -7.1667, A 0.000, B 0.000, C 0.000 }
gfCNCPoint5[11515] = {X 347.9624, Y 31.9018, Z -7.1667, A 0.000, B 0.000, C 0.000 }
gfCNCPoint5[11516] = {X 348.6980, Y 31.6161, Z -7.1667, A 0.000, B 0.000, C 0.000 }
gfCNCPoint5[11517] = {X 349.3519, Y 31.1743, Z -7.1667, A 0.000, B 0.000, C 0.000 }
gfCNCPoint5[11518] = {X 350.1526, Y 30.3709, Z -7.1667, A 0.000, B 0.000, C 0.000 }
gfCNCPoint5[11519] = {X 350.8131, Y 29.4487, Z -7.1667, A 0.000, B 0.000, C 0.000 }
gfCNCPoint5[11520] = {X 351.3161, Y 28.4320, Z -7.1667, A 0.000, B 0.000, C 0.000 }
gfCNCPoint5[11521] = {X 351.6482, Y 27.3474, Z -7.1667, A 0.000, B 0.000, C 0.000 }
gfCNCPoint5[11522] = {X 351.8767, Y 25.7621, Z -7.1667, A 0.000, B 0.000, C 0.000 }
gfCNCPoint5[11523] = {X 351.9020, Y 24.1607, Z -7.1667, A 0.000, B 0.000, C 0.000 }
gfCNCPoint5[11524] = {X 351.7237, Y 22.5690, Z -7.1667, A 0.000, B 0.000, C 0.000 }
gfCNCPoint5[11525] = {X 351.4417, Y 21.4556, Z -7.1667, A 0.000, B 0.000, C 0.000 }
gfCNCPoint5[11526] = {X 350.9675, Y 20.4095, Z -7.1667, A 0.000, B 0.000, C 0.000 }
gfCNCPoint5[11527] = {X 350.3160, Y 19.4636, Z -7.1667, A 0.000, B 0.000, C 0.000 }
gfCNCPoint5[11528] = {X 349.6854, Y 18.8479, Z -7.1667, A 0.000, B 0.000, C 0.000 }
gfCNCPoint5[11529] = {X 348.9297, Y 18.3944, Z -7.1667, A 0.000, B 0.000, C 0.000 }
gfCNCPoint5[11530] = {X 348.0896, Y 18.1279, Z -7.1667, A 0.000, B 0.000, C 0.000 }
gfCNCPoint5[11531] = {X 346.9970, Y 17.9940, Z -7.1667, A 0.000, B 0.000, C 0.000 }
gfCNCPoint5[11532] = {X 345.8964, Y 18.0114, Z -7.1667, A 0.000, B 0.000, C 0.000 }
gfCNCPoint5[11533] = {X 344.8086, Y 18.1797, Z -7.1667, A 0.000, B 0.000, C 0.000 }
gfCNCPoint5[11534] = {X 343.7542, Y 18.4957, Z -7.1667, A 0.000, B 0.000, C 0.000 }
gfCNCPoint5[11535] = {X 343.3272, Y 19.5039, Z -7.1667, A 0.000, B 0.000, C 0.000 }
gfCNCPoint5[11536] = {X 342.7891, Y 20.4574, Z -7.1667, A 0.000, B 0.000, C 0.000 }
gfCNCPoint5[11537] = {X 342.1467, Y 21.3441, Z -7.1667, A 0.000, B 0.000, C 0.000 }
gfCNCPoint5[11538] = {X 340.2859, Y 19.8284, Z -7.1667, A 0.000, B 0.000, C 0.000 }
gfCNCPoint5[11539] = {X 339.6798, Y 20.4856, Z -7.1667, A 0.000, B 0.000, C 0.000 }
gfCNCPoint5[11540] = {X 338.9976, Y 21.0636, Z -7.1667, A 0.000, B 0.000, C 0.000 }
gfCNCPoint5[11541] = {X 338.2497, Y 21.6141, Z -7.1667, A 0.000, B 0.000, C 0.000 }
gfCNCPoint5[11542] = {X 337.8538, Y 21.8795, Z -7.1667, A 0.000, B 0.000, C 0.000 }
gfCNCPoint5[11543] = {X 337.4413, Y 22.1185, Z -7.1667, A 0.000, B 0.000, C 0.000 }
gfCNCPoint5[11544] = {X 336.3239, Y 22.6023, Z -7.1667, A 0.000, B 0.000, C 0.000 }
gfCNCPoint5[11545] = {X 335.1415, Y 22.8932, Z -7.1667, A 0.000, B 0.000, C 0.000 }
gfCNCPoint5[11546] = {X 333.9271, Y 22.9829, Z -7.1667, A 0.000, B 0.000, C 0.000 }
gfCNCPoint5[11547] = {X 332.7148, Y 22.8690, Z -7.1667, A 0.000, B 0.000, C 0.000 }
gfCNCPoint5[11548] = {X 331.5384, Y 22.5546, Z -7.1667, A 0.000, B 0.000, C 0.000 }
gfCNCPoint5[11549] = {X 330.4309, Y 22.0485, Z -7.1667, A 0.000, B 0.000, C 0.000 }
gfCNCPoint5[11550] = {X 329.5143, Y 21.4374, Z -7.1667, A 0.000, B 0.000, C 0.000 }
gfCNCPoint5[11551] = {X 328.7005, Y 20.6949, Z -7.1667, A 0.000, B 0.000, C 0.000 }
gfCNCPoint5[11552] = {X 328.0080, Y 19.8382, Z -7.1667, A 0.000, B 0.000, C 0.000 }
gfCNCPoint5[11553] = {X 327.4528, Y 18.8869, Z -7.1667, A 0.000, B 0.000, C 0.000 }
gfCNCPoint5[11554] = {X 323.9321, Y 11.6443, Z -7.1667, A 0.000, B 0.000, C 0.000 }
gfCNCPoint5[11555] = {X 323.5337, Y 10.6421, Z -7.1667, A 0.000, B 0.000, C 0.000 }
gfCNCPoint5[11556] = {X 323.2878, Y 9.5921, Z -7.1667, A 0.000, B 0.000, C 0.000 }
gfCNCPoint5[11557] = {X 323.1997, Y 8.5173, Z -7.1667, A 0.000, B 0.000, C 0.000 }
gfCNCPoint5[11558] = {X 323.2713, Y 7.4412, Z -7.1667, A 0.000, B 0.000, C 0.000 }
gfCNCPoint5[11559] = {X 323.4720, Y 6.4883, Z -7.1667, A 0.000, B 0.000, C 0.000 }
gfCNCPoint5[11560] = {X 323.7980, Y 5.5707, Z -7.1667, A 0.000, B 0.000, C 0.000 }
gfCNCPoint5[11561] = {X 324.2436, Y 4.7049, Z -7.1667, A 0.000, B 0.000, C 0.000 }
gfCNCPoint5[11562] = {X 168.0206, Y 4.7049, Z -7.1667, A 0.000, B 0.000, C 0.000 }
gfCNCPoint5[11563] = {X 168.0206, Y 9.5049, Z -7.1667, A 0.000, B 0.000, C 0.000 }
gfCNCPoint5[11564] = {X 166.5360, Y 9.5049, Z -7.1667, A 0.000, B 0.000, C 0.000 }
gfCNCPoint5[11565] = {X 166.5855, Y 9.9931, Z -7.1667, A 0.000, B 0.000, C 0.000 }
gfCNCPoint5[11566] = {X 166.6021, Y 10.4835, Z -7.1667, A 0.000, B 0.000, C 0.000 }
gfCNCPoint5[11567] = {X 166.6021, Y 13.0969, Z -7.1667, A 0.000, B 0.000, C 0.000 }
gfCNCPoint5[11568] = {X 166.8569, Y 11.8209, Z -7.1667, A 0.000, B 0.000, C 0.000 }
gfCNCPoint5[11569] = {X 167.3349, Y 10.6107, Z -7.1667, A 0.000, B 0.000, C 0.000 }
gfCNCPoint5[11570] = {X 168.0206, Y 9.5049, Z -7.1667, A 0.000, B 0.000, C 0.000 }
gfCNCPoint5[11571] = {X 168.0206, Y 7.1049, Z -7.1667, A 0.000, B 0.000, C 0.000 }
gfCNCPoint5[11572] = {X 162.8433, Y 7.1049, Z -7.1667, A 0.000, B 0.000, C 0.000 }
gfCNCPoint5[11573] = {X 163.4702, Y 7.9130, Z -7.1667, A 0.000, B 0.000, C 0.000 }
gfCNCPoint5[11574] = {X 163.9149, Y 8.8340, Z -7.1667, A 0.000, B 0.000, C 0.000 }
gfCNCPoint5[11575] = {X 164.1578, Y 9.8275, Z -7.1667, A 0.000, B 0.000, C 0.000 }
gfCNCPoint5[11576] = {X 164.1910, Y 10.1548, Z -7.1667, A 0.000, B 0.000, C 0.000 }
gfCNCPoint5[11577] = {X 164.2021, Y 10.4835, Z -7.1667, A 0.000, B 0.000, C 0.000 }
gfCNCPoint5[11578] = {X 164.2021, Y 17.4615, Z -7.1667, A 0.000, B 0.000, C 0.000 }
gfCNCPoint5[11579] = {X 164.1140, Y 18.3847, Z -7.1667, A 0.000, B 0.000, C 0.000 }
gfCNCPoint5[11580] = {X 163.8528, Y 19.2745, Z -7.1667, A 0.000, B 0.000, C 0.000 }
gfCNCPoint5[11581] = {X 163.4280, Y 20.0989, Z -7.1667, A 0.000, B 0.000, C 0.000 }
gfCNCPoint5[11582] = {X 162.8550, Y 20.8280, Z -7.1667, A 0.000, B 0.000, C 0.000 }
gfCNCPoint5[11583] = {X 162.1544, Y 21.4355, Z -7.1667, A 0.000, B 0.000, C 0.000 }
gfCNCPoint5[11584] = {X 161.3514, Y 21.8996, Z -7.1667, A 0.000, B 0.000, C 0.000 }
gfCNCPoint5[11585] = {X 160.4752, Y 22.2033, Z -7.1667, A 0.000, B 0.000, C 0.000 }
gfCNCPoint5[11586] = {X 162.1766, Y 29.1994, Z -7.1667, A 0.000, B 0.000, C 0.000 }
gfCNCPoint5[11587] = {X 161.1139, Y 29.4079, Z -7.1667, A 0.000, B 0.000, C 0.000 }
gfCNCPoint5[11588] = {X 160.0367, Y 29.5204, Z -7.1667, A 0.000, B 0.000, C 0.000 }
gfCNCPoint5[11589] = {X 160.0362, Y 38.3363, Z -7.1667, A 0.000, B 0.000, C 0.000 }
gfCNCPoint5[11590] = {X 160.6844, Y 39.6935, Z -7.1667, A 0.000, B 0.000, C 0.000 }
gfCNCPoint5[11591] = {X 161.1592, Y 41.1206, Z -7.1667, A 0.000, B 0.000, C 0.000 }
gfCNCPoint5[11592] = {X 162.0521, Y 41.1205, Z -7.1667, A 0.000, B 0.000, C 0.000 }
gfCNCPoint5[11593] = {X 161.8698, Y 40.3467, Z -7.1667, A 0.000, B 0.000, C 0.000 }
gfCNCPoint5[11594] = {X 161.7172, Y 39.5665, Z -7.1667, A 0.000, B 0.000, C 0.000 }
gfCNCPoint5[11595] = {X 161.5939, Y 38.7921, Z -7.1667, A 0.000, B 0.000, C 0.000 }
gfCNCPoint5[11596] = {X 161.3797, Y 36.8677, Z -7.1667, A 0.000, B 0.000, C 0.000 }
gfCNCPoint5[11597] = {X 161.3311, Y 34.9320, Z -7.1667, A 0.000, B 0.000, C 0.000 }
gfCNCPoint5[11598] = {X 161.4485, Y 32.9993, Z -7.1667, A 0.000, B 0.000, C 0.000 }
gfCNCPoint5[11599] = {X 161.7311, Y 31.0837, Z -7.1667, A 0.000, B 0.000, C 0.000 }
gfCNCPoint5[11600] = {X 162.1766, Y 29.1994, Z -7.1667, A 0.000, B 0.000, C 0.000 }
gfCNCPoint5[11601] = {X 161.6095, Y 26.8674, Z -7.1667, A 0.000, B 0.000, C 0.000 }
gfCNCPoint5[11602] = {X 160.4740, Y 27.0728, Z -7.1667, A 0.000, B 0.000, C 0.000 }
gfCNCPoint5[11603] = {X 159.3221, Y 27.1415, Z -7.1667, A 0.000, B 0.000, C 0.000 }
gfCNCPoint5[11604] = {X 158.6609, Y 27.1415, Z -7.1667, A 0.000, B 0.000, C 0.000 }
gfCNCPoint5[11605] = {X 158.1481, Y 27.1262, Z -7.1667, A 0.000, B 0.000, C 0.000 }
gfCNCPoint5[11606] = {X 157.6368, Y 27.0838, Z -7.1667, A 0.000, B 0.000, C 0.000 }
gfCNCPoint5[11607] = {X 157.6362, Y 38.9959, Z -7.1667, A 0.000, B 0.000, C 0.000 }
gfCNCPoint5[11608] = {X 158.2201, Y 40.0482, Z -7.1667, A 0.000, B 0.000, C 0.000 }
gfCNCPoint5[11609] = {X 158.6692, Y 41.1647, Z -7.1667, A 0.000, B 0.000, C 0.000 }
gfCNCPoint5[11610] = {X 158.9767, Y 42.3283, Z -7.1667, A 0.000, B 0.000, C 0.000 }
gfCNCPoint5[11611] = {X 159.1378, Y 43.5209, Z -7.1667, A 0.000, B 0.000, C 0.000 }
gfCNCPoint5[11612] = {X 165.4260, Y 43.5200, Z -7.1667, A 0.000, B 0.000, C 0.000 }
gfCNCPoint5[11613] = {X 164.8369, Y 42.0454, Z -7.1667, A 0.000, B 0.000, C 0.000 }
gfCNCPoint5[11614] = {X 164.3772, Y 40.5255, Z -7.1667, A 0.000, B 0.000, C 0.000 }
gfCNCPoint5[11615] = {X 164.2179, Y 39.8500, Z -7.1667, A 0.000, B 0.000, C 0.000 }
gfCNCPoint5[11616] = {X 164.0841, Y 39.1688, Z -7.1667, A 0.000, B 0.000, C 0.000 }
gfCNCPoint5[11617] = {X 163.9649, Y 38.4200, Z -7.1667, A 0.000, B 0.000, C 0.000 }
gfCNCPoint5[11618] = {X 163.7492, Y 36.2691, Z -7.1667, A 0.000, B 0.000, C 0.000 }
gfCNCPoint5[11619] = {X 163.7648, Y 34.1076, Z -7.1667, A 0.000, B 0.000, C 0.000 }
gfCNCPoint5[11620] = {X 164.0115, Y 31.9601, Z -7.1667, A 0.000, B 0.000, C 0.000 }
gfCNCPoint5[11621] = {X 164.4864, Y 29.8513, Z -7.1667, A 0.000, B 0.000, C 0.000 }
gfCNCPoint5[11622] = {X 164.8367, Y 28.7351, Z -7.1667, A 0.000, B 0.000, C 0.000 }
gfCNCPoint5[11623] = {X 165.2510, Y 27.6411, Z -7.1667, A 0.000, B 0.000, C 0.000 }
gfCNCPoint5[11624] = {X 165.8679, Y 26.3082, Z -7.1667, A 0.000, B 0.000, C 0.000 }
gfCNCPoint5[11625] = {X 166.6028, Y 25.0367, Z -7.1667, A 0.000, B 0.000, C 0.000 }
gfCNCPoint5[11626] = {X 167.4498, Y 23.8368, Z -7.1667, A 0.000, B 0.000, C 0.000 }
gfCNCPoint5[11627] = {X 167.1640, Y 23.1367, Z -7.1667, A 0.000, B 0.000, C 0.000 }
gfCNCPoint5[11628] = {X 166.2875, Y 24.1835, Z -7.1667, A 0.000, B 0.000, C 0.000 }
gfCNCPoint5[11629] = {X 165.2726, Y 25.0966, Z -7.1667, A 0.000, B 0.000, C 0.000 }
gfCNCPoint5[11630] = {X 164.1392, Y 25.8578, Z -7.1667, A 0.000, B 0.000, C 0.000 }
gfCNCPoint5[11631] = {X 162.9100, Y 26.4520, Z -7.1667, A 0.000, B 0.000, C 0.000 }
gfCNCPoint5[11632] = {X 161.6095, Y 26.8674, Z -7.1667, A 0.000, B 0.000, C 0.000 }
gfCNCPoint5[11633] = {X 161.0424, Y 24.5354, Z -7.1667, A 0.000, B 0.000, C 0.000 }
gfCNCPoint5[11634] = {X 160.1884, Y 24.6898, Z -7.1667, A 0.000, B 0.000, C 0.000 }
gfCNCPoint5[11635] = {X 159.3221, Y 24.7415, Z -7.1667, A 0.000, B 0.000, C 0.000 }
gfCNCPoint5[11636] = {X 158.6691, Y 24.7415, Z -7.1667, A 0.000, B 0.000, C 0.000 }
gfCNCPoint5[11637] = {X 158.2831, Y 24.7300, Z -7.1667, A 0.000, B 0.000, C 0.000 }
gfCNCPoint5[11638] = {X 157.8982, Y 24.6981, Z -7.1667, A 0.000, B 0.000, C 0.000 }
gfCNCPoint5[11639] = {X 156.9783, Y 24.5373, Z -7.1667, A 0.000, B 0.000, C 0.000 }
gfCNCPoint5[11640] = {X 156.0863, Y 24.2605, Z -7.1667, A 0.000, B 0.000, C 0.000 }
gfCNCPoint5[11641] = {X 155.2370, Y 23.8723, Z -7.1667, A 0.000, B 0.000, C 0.000 }
gfCNCPoint5[11642] = {X 155.2362, Y 39.7518, Z -7.1667, A 0.000, B 0.000, C 0.000 }
gfCNCPoint5[11643] = {X 155.8269, Y 40.6434, Z -7.1667, A 0.000, B 0.000, C 0.000 }
gfCNCPoint5[11644] = {X 156.2811, Y 41.6117, Z -7.1667, A 0.000, B 0.000, C 0.000 }
gfCNCPoint5[11645] = {X 156.5890, Y 42.6359, Z -7.1667, A 0.000, B 0.000, C 0.000 }
gfCNCPoint5[11646] = {X 156.7441, Y 43.6941, Z -7.1667, A 0.000, B 0.000, C 0.000 }
gfCNCPoint5[11647] = {X 156.7579, Y 43.9463, Z -7.1667, A 0.000, B 0.000, C 0.000 }
gfCNCPoint5[11648] = {X 156.7631, Y 44.1988, Z -7.1667, A 0.000, B 0.000, C 0.000 }
gfCNCPoint5[11649] = {X 156.7628, Y 45.0700, Z -7.1667, A 0.000, B 0.000, C 0.000 }
gfCNCPoint5[11650] = {X 156.7347, Y 45.6426, Z -7.1667, A 0.000, B 0.000, C 0.000 }
gfCNCPoint5[11651] = {X 156.6616, Y 46.2112, Z -7.1667, A 0.000, B 0.000, C 0.000 }
gfCNCPoint5[11652] = {X 157.9054, Y 46.0005, Z -7.1667, A 0.000, B 0.000, C 0.000 }
gfCNCPoint5[11653] = {X 159.1643, Y 45.9207, Z -7.1667, A 0.000, B 0.000, C 0.000 }
gfCNCPoint5[11654] = {X 159.2312, Y 45.9202, Z -7.1667, A 0.000, B 0.000, C 0.000 }
gfCNCPoint5[11655] = {X 159.2980, Y 45.9200, Z -7.1667, A 0.000, B 0.000, C 0.000 }
gfCNCPoint5[11656] = {X 169.6790, Y 45.9200, Z -7.1667, A 0.000, B 0.000, C 0.000 }
gfCNCPoint5[11657] = {X 168.8979, Y 44.8498, Z -7.1667, A 0.000, B 0.000, C 0.000 }
gfCNCPoint5[11658] = {X 168.2080, Y 43.7186, Z -7.1667, A 0.000, B 0.000, C 0.000 }
gfCNCPoint5[11659] = {X 167.6142, Y 42.5342, Z -7.1667, A 0.000, B 0.000, C 0.000 }
gfCNCPoint5[11660] = {X 167.1234, Y 41.3128, Z -7.1667, A 0.000, B 0.000, C 0.000 }
gfCNCPoint5[11661] = {X 166.7347, Y 40.0551, Z -7.1667, A 0.000, B 0.000, C 0.000 }
gfCNCPoint5[11662] = {X 166.4508, Y 38.7698, Z -7.1667, A 0.000, B 0.000, C 0.000 }
gfCNCPoint5[11663] = {X 166.3359, Y 38.0481, Z -7.1667, A 0.000, B 0.000, C 0.000 }
gfCNCPoint5[11664] = {X 166.1450, Y 36.1220, Z -7.1667, A 0.000, B 0.000, C 0.000 }
gfCNCPoint5[11665] = {X 166.1646, Y 34.1866, Z -7.1667, A 0.000, B 0.000, C 0.000 }
gfCNCPoint5[11666] = {X 166.3943, Y 32.2648, Z -7.1667, A 0.000, B 0.000, C 0.000 }
gfCNCPoint5[11667] = {X 166.8316, Y 30.3794, Z -7.1667, A 0.000, B 0.000, C 0.000 }
gfCNCPoint5[11668] = {X 167.4712, Y 28.5526, Z -7.1667, A 0.000, B 0.000, C 0.000 }
gfCNCPoint5[11669] = {X 168.2319, Y 26.9822, Z -7.1667, A 0.000, B 0.000, C 0.000 }
gfCNCPoint5[11670] = {X 169.1845, Y 25.5203, Z -7.1667, A 0.000, B 0.000, C 0.000 }
gfCNCPoint5[11671] = {X 170.3138, Y 24.1902, Z -7.1667, A 0.000, B 0.000, C 0.000 }
gfCNCPoint5[11672] = {X 169.9863, Y 23.6219, Z -7.1667, A 0.000, B 0.000, C 0.000 }
gfCNCPoint5[11673] = {X 169.7113, Y 23.0264, Z -7.1667, A 0.000, B 0.000, C 0.000 }
gfCNCPoint5[11674] = {X 167.1001, Y 16.6309, Z -7.1667, A 0.000, B 0.000, C 0.000 }
gfCNCPoint5[11675] = {X 166.7820, Y 15.6636, Z -7.1667, A 0.000, B 0.000, C 0.000 }
gfCNCPoint5[11676] = {X 166.6021, Y 14.6613, Z -7.1667, A 0.000, B 0.000, C 0.000 }
gfCNCPoint5[11677] = {X 166.6021, Y 17.4615, Z -7.1667, A 0.000, B 0.000, C 0.000 }
gfCNCPoint5[11678] = {X 166.5130, Y 18.5970, Z -7.1667, A 0.000, B 0.000, C 0.000 }
gfCNCPoint5[11679] = {X 166.2479, Y 19.7047, Z -7.1667, A 0.000, B 0.000, C 0.000 }
gfCNCPoint5[11680] = {X 165.8132, Y 20.7575, Z -7.1667, A 0.000, B 0.000, C 0.000 }
gfCNCPoint5[11681] = {X 165.2197, Y 21.7296, Z -7.1667, A 0.000, B 0.000, C 0.000 }
gfCNCPoint5[11682] = {X 164.3789, Y 22.6986, Z -7.1667, A 0.000, B 0.000, C 0.000 }
gfCNCPoint5[11683] = {X 163.3812, Y 23.5049, Z -7.1667, A 0.000, B 0.000, C 0.000 }
gfCNCPoint5[11684] = {X 162.2573, Y 24.1236, Z -7.1667, A 0.000, B 0.000, C 0.000 }
gfCNCPoint5[11685] = {X 161.0424, Y 24.5354, Z -7.1667, A 0.000, B 0.000, C 0.000 }
gfCNCPoint5[11686] = {X 160.4752, Y 22.2033, Z -7.1667, A 0.000, B 0.000, C 0.000 }
gfCNCPoint5[11687] = {X 159.9028, Y 22.3069, Z -7.1667, A 0.000, B 0.000, C 0.000 }
gfCNCPoint5[11688] = {X 159.3221, Y 22.3415, Z -7.1667, A 0.000, B 0.000, C 0.000 }
gfCNCPoint5[11689] = {X 158.6774, Y 22.3415, Z -7.1667, A 0.000, B 0.000, C 0.000 }
gfCNCPoint5[11690] = {X 157.8805, Y 22.2736, Z -7.1667, A 0.000, B 0.000, C 0.000 }
gfCNCPoint5[11691] = {X 157.1052, Y 22.0773, Z -7.1667, A 0.000, B 0.000, C 0.000 }
gfCNCPoint5[11692] = {X 156.3721, Y 21.7577, Z -7.1667, A 0.000, B 0.000, C 0.000 }
gfCNCPoint5[11693] = {X 155.5228, Y 21.1799, Z -7.1667, A 0.000, B 0.000, C 0.000 }
gfCNCPoint5[11694] = {X 154.8123, Y 20.4380, Z -7.1667, A 0.000, B 0.000, C 0.000 }
gfCNCPoint5[11695] = {X 152.8371, Y 20.4387, Z -7.1667, A 0.000, B 0.000, C 0.000 }
gfCNCPoint5[11696] = {X 152.8361, Y 40.6543, Z -7.1667, A 0.000, B 0.000, C 0.000 }
gfCNCPoint5[11697] = {X 153.1746, Y 41.0203, Z -7.1667, A 0.000, B 0.000, C 0.000 }
gfCNCPoint5[11698] = {X 153.6801, Y 41.7247, Z -7.1667, A 0.000, B 0.000, C 0.000 }
gfCNCPoint5[11699] = {X 154.0538, Y 42.5070, Z -7.1667, A 0.000, B 0.000, C 0.000 }
gfCNCPoint5[11700] = {X 154.2838, Y 43.3429, Z -7.1667, A 0.000, B 0.000, C 0.000 }
gfCNCPoint5[11701] = {X 154.3631, Y 44.2062, Z -7.1667, A 0.000, B 0.000, C 0.000 }
gfCNCPoint5[11702] = {X 154.3629, Y 45.0469, Z -7.1667, A 0.000, B 0.000, C 0.000 }
gfCNCPoint5[11703] = {X 154.3440, Y 45.4308, Z -7.1667, A 0.000, B 0.000, C 0.000 }
gfCNCPoint5[11704] = {X 154.2951, Y 45.8119, Z -7.1667, A 0.000, B 0.000, C 0.000 }
gfCNCPoint5[11705] = {X 154.0370, Y 46.7541, Z -7.1667, A 0.000, B 0.000, C 0.000 }
gfCNCPoint5[11706] = {X 153.5963, Y 47.6260, Z -7.1667, A 0.000, B 0.000, C 0.000 }
gfCNCPoint5[11707] = {X 152.9909, Y 48.3926, Z -7.1667, A 0.000, B 0.000, C 0.000 }
gfCNCPoint5[11708] = {X 152.2448, Y 49.0233, Z -7.1667, A 0.000, B 0.000, C 0.000 }
gfCNCPoint5[11709] = {X 151.3881, Y 49.4928, Z -7.1667, A 0.000, B 0.000, C 0.000 }
gfCNCPoint5[11710] = {X 150.4551, Y 49.7822, Z -7.1667, A 0.000, B 0.000, C 0.000 }
gfCNCPoint5[11711] = {X 149.4831, Y 49.8800, Z -7.1667, A 0.000, B 0.000, C 0.000 }
gfCNCPoint5[11712] = {X 143.0396, Y 49.8800, Z -7.1667, A 0.000, B 0.000, C 0.000 }
gfCNCPoint5[11713] = {X 142.0923, Y 49.7872, Z -7.1667, A 0.000, B 0.000, C 0.000 }
gfCNCPoint5[11714] = {X 141.1811, Y 49.5122, Z -7.1667, A 0.000, B 0.000, C 0.000 }
gfCNCPoint5[11715] = {X 140.3405, Y 49.0656, Z -7.1667, A 0.000, B 0.000, C 0.000 }
gfCNCPoint5[11716] = {X 139.6026, Y 48.4643, Z -7.1667, A 0.000, B 0.000, C 0.000 }
gfCNCPoint5[11717] = {X 138.9955, Y 47.7312, Z -7.1667, A 0.000, B 0.000, C 0.000 }
gfCNCPoint5[11718] = {X 138.5423, Y 46.8942, Z -7.1667, A 0.000, B 0.000, C 0.000 }
gfCNCPoint5[11719] = {X 138.2601, Y 45.9852, Z -7.1667, A 0.000, B 0.000, C 0.000 }
gfCNCPoint5[11720] = {X 138.1598, Y 45.0386, Z -7.1667, A 0.000, B 0.000, C 0.000 }
gfCNCPoint5[11721] = {X 138.1601, Y 44.1417, Z -7.1667, A 0.000, B 0.000, C 0.000 }
gfCNCPoint5[11722] = {X 138.2148, Y 43.4769, Z -7.1667, A 0.000, B 0.000, C 0.000 }
gfCNCPoint5[11723] = {X 138.3597, Y 42.8258, Z -7.1667, A 0.000, B 0.000, C 0.000 }
gfCNCPoint5[11724] = {X 129.1532, Y 40.1052, Z -7.1667, A 0.000, B 0.000, C 0.000 }
gfCNCPoint5[11725] = {X 129.5665, Y 38.9035, Z -7.1667, A 0.000, B 0.000, C 0.000 }
gfCNCPoint5[11726] = {X 130.0836, Y 37.7426, Z -7.1667, A 0.000, B 0.000, C 0.000 }
gfCNCPoint5[11727] = {X 130.0836, Y 31.6021, Z -7.1667, A 0.000, B 0.000, C 0.000 }
gfCNCPoint5[11728] = {X 129.2065, Y 31.3798, Z -7.1667, A 0.000, B 0.000, C 0.000 }
gfCNCPoint5[11729] = {X 128.3450, Y 31.1031, Z -7.1667, A 0.000, B 0.000, C 0.000 }
gfCNCPoint5[11730] = {X 128.3450, Y 38.3307, Z -7.1667, A 0.000, B 0.000, C 0.000 }
gfCNCPoint5[11731] = {X 128.7850, Y 39.2016, Z -7.1667, A 0.000, B 0.000, C 0.000 }
gfCNCPoint5[11732] = {X 129.1532, Y 40.1052, Z -7.1667, A 0.000, B 0.000, C 0.000 }
gfCNCPoint5[11733] = {X 131.4548, Y 40.7854, Z -7.1667, A 0.000, B 0.000, C 0.000 }
gfCNCPoint5[11734] = {X 131.9017, Y 39.5320, Z -7.1667, A 0.000, B 0.000, C 0.000 }
gfCNCPoint5[11735] = {X 132.4836, Y 38.3354, Z -7.1667, A 0.000, B 0.000, C 0.000 }
gfCNCPoint5[11736] = {X 132.4836, Y 29.5202, Z -7.1667, A 0.000, B 0.000, C 0.000 }
gfCNCPoint5[11737] = {X 131.3527, Y 29.3994, Z -7.1667, A 0.000, B 0.000, C 0.000 }
gfCNCPoint5[11738] = {X 130.2381, Y 29.1726, Z -7.1667, A 0.000, B 0.000, C 0.000 }
gfCNCPoint5[11739] = {X 129.1498, Y 28.8421, Z -7.1667, A 0.000, B 0.000, C 0.000 }
gfCNCPoint5[11740] = {X 128.0254, Y 28.3768, Z -7.1667, A 0.000, B 0.000, C 0.000 }
gfCNCPoint5[11741] = {X 126.9536, Y 27.8008, Z -7.1667, A 0.000, B 0.000, C 0.000 }
gfCNCPoint5[11742] = {X 125.9451, Y 27.1199, Z -7.1667, A 0.000, B 0.000, C 0.000 }
gfCNCPoint5[11743] = {X 125.9450, Y 38.9911, Z -7.1667, A 0.000, B 0.000, C 0.000 }
gfCNCPoint5[11744] = {X 126.4742, Y 39.9293, Z -7.1667, A 0.000, B 0.000, C 0.000 }
gfCNCPoint5[11745] = {X 126.8960, Y 40.9205, Z -7.1667, A 0.000, B 0.000, C 0.000 }
gfCNCPoint5[11746] = {X 127.2098, Y 41.9730, Z -7.1667, A 0.000, B 0.000, C 0.000 }
gfCNCPoint5[11747] = {X 127.4025, Y 43.0542, Z -7.1667, A 0.000, B 0.000, C 0.000 }
gfCNCPoint5[11748] = {X 127.4714, Y 44.1502, Z -7.1667, A 0.000, B 0.000, C 0.000 }
gfCNCPoint5[11749] = {X 127.4716, Y 45.0000, Z -7.1667, A 0.000, B 0.000, C 0.000 }
gfCNCPoint5[11750] = {X 127.4070, Y 46.1159, Z -7.1667, A 0.000, B 0.000, C 0.000 }
gfCNCPoint5[11751] = {X 127.2143, Y 47.2168, Z -7.1667, A 0.000, B 0.000, C 0.000 }
gfCNCPoint5[11752] = {X 126.8960, Y 48.2883, Z -7.1667, A 0.000, B 0.000, C 0.000 }
gfCNCPoint5[11753] = {X 126.2883, Y 49.6376, Z -7.1667, A 0.000, B 0.000, C 0.000 }
gfCNCPoint5[11754] = {X 125.4821, Y 50.8786, Z -7.1667, A 0.000, B 0.000, C 0.000 }
gfCNCPoint5[11755] = {X 124.4962, Y 51.9821, Z -7.1667, A 0.000, B 0.000, C 0.000 }
gfCNCPoint5[11756] = {X 123.3536, Y 52.9225, Z -7.1667, A 0.000, B 0.000, C 0.000 }
gfCNCPoint5[11757] = {X 122.0810, Y 53.6778, Z -7.1667, A 0.000, B 0.000, C 0.000 }
gfCNCPoint5[11758] = {X 120.7081, Y 54.2302, Z -7.1667, A 0.000, B 0.000, C 0.000 }
gfCNCPoint5[11759] = {X 119.2671, Y 54.5669, Z -7.1667, A 0.000, B 0.000, C 0.000 }
gfCNCPoint5[11760] = {X 117.7916, Y 54.6800, Z -7.1667, A 0.000, B 0.000, C 0.000 }
gfCNCPoint5[11761] = {X 111.9185, Y 54.6800, Z -7.1667, A 0.000, B 0.000, C 0.000 }
gfCNCPoint5[11762] = {X 111.7443, Y 54.6784, Z -7.1667, A 0.000, B 0.000, C 0.000 }
gfCNCPoint5[11763] = {X 111.5702, Y 54.6737, Z -7.1667, A 0.000, B 0.000, C 0.000 }
gfCNCPoint5[11764] = {X 111.0521, Y 69.0644, Z -7.1667, A 0.000, B 0.000, C 0.000 }
gfCNCPoint5[11765] = {X 109.0264, Y 68.9057, Z -7.1667, A 0.000, B 0.000, C 0.000 }
gfCNCPoint5[11766] = {X 107.0213, Y 68.5768, Z -7.1667, A 0.000, B 0.000, C 0.000 }
gfCNCPoint5[11767] = {X 105.0765, Y 68.8983, Z -7.1667, A 0.000, B 0.000, C 0.000 }
gfCNCPoint5[11768] = {X 103.1119, Y 69.0597, Z -7.1667, A 0.000, B 0.000, C 0.000 }
gfCNCPoint5[11769] = {X 101.1407, Y 69.0599, Z -7.1667, A 0.000, B 0.000, C 0.000 }
gfCNCPoint5[11770] = {X 99.1761, Y 68.8989, Z -7.1667, A 0.000, B 0.000, C 0.000 }
gfCNCPoint5[11771] = {X 97.2313, Y 68.5777, Z -7.1667, A 0.000, B 0.000, C 0.000 }
gfCNCPoint5[11772] = {X 95.6131, Y 68.8563, Z -7.1667, A 0.000, B 0.000, C 0.000 }
gfCNCPoint5[11773] = {X 93.9796, Y 69.0240, Z -7.1667, A 0.000, B 0.000, C 0.000 }
gfCNCPoint5[11774] = {X 92.3385, Y 69.0800, Z -7.1667, A 0.000, B 0.000, C 0.000 }
gfCNCPoint5[11775] = {X 86.6884, Y 69.0800, Z -7.1667, A 0.000, B 0.000, C 0.000 }
gfCNCPoint5[11776] = {X 84.7315, Y 70.2669, Z -7.1667, A 0.000, B 0.000, C 0.000 }
gfCNCPoint5[11777] = {X 82.6868, Y 71.2951, Z -7.1667, A 0.000, B 0.000, C 0.000 }
gfCNCPoint5[11778] = {X 107.2670, Y 71.2951, Z -7.1667, A 0.000, B 0.000, C 0.000 }
gfCNCPoint5[11779] = {X 109.1203, Y 70.1132, Z -7.1667, A 0.000, B 0.000, C 0.000 }
gfCNCPoint5[11780] = {X 111.0521, Y 69.0644, Z -7.1667, A 0.000, B 0.000, C 0.000 }
gfCNCPoint5[11781] = {X 111.1384, Y 66.6660, Z -7.1667, A 0.000, B 0.000, C 0.000 }
gfCNCPoint5[11782] = {X 109.0667, Y 66.4916, Z -7.1667, A 0.000, B 0.000, C 0.000 }
gfCNCPoint5[11783] = {X 107.0213, Y 66.1197, Z -7.1667, A 0.000, B 0.000, C 0.000 }
gfCNCPoint5[11784] = {X 105.0796, Y 66.4776, Z -7.1667, A 0.000, B 0.000, C 0.000 }
gfCNCPoint5[11785] = {X 103.1135, Y 66.6574, Z -7.1667, A 0.000, B 0.000, C 0.000 }
gfCNCPoint5[11786] = {X 101.1392, Y 66.6576, Z -7.1667, A 0.000, B 0.000, C 0.000 }
gfCNCPoint5[11787] = {X 99.1730, Y 66.4782, Z -7.1667, A 0.000, B 0.000, C 0.000 }
gfCNCPoint5[11788] = {X 97.2313, Y 66.1207, Z -7.1667, A 0.000, B 0.000, C 0.000 }
gfCNCPoint5[11789] = {X 95.6161, Y 66.4308, Z -7.1667, A 0.000, B 0.000, C 0.000 }
gfCNCPoint5[11790] = {X 93.9821, Y 66.6176, Z -7.1667, A 0.000, B 0.000, C 0.000 }
gfCNCPoint5[11791] = {X 92.3385, Y 66.6800, Z -7.1667, A 0.000, B 0.000, C 0.000 }
gfCNCPoint5[11792] = {X 85.9487, Y 66.6800, Z -7.1667, A 0.000, B 0.000, C 0.000 }
gfCNCPoint5[11793] = {X 83.8778, Y 67.9936, Z -7.1667, A 0.000, B 0.000, C 0.000 }
gfCNCPoint5[11794] = {X 81.6944, Y 69.1099, Z -7.1667, A 0.000, B 0.000, C 0.000 }
gfCNCPoint5[11795] = {X 79.6014, Y 69.9548, Z -7.1667, A 0.000, B 0.000, C 0.000 }
gfCNCPoint5[11796] = {X 77.4441, Y 70.6185, Z -7.1667, A 0.000, B 0.000, C 0.000 }
gfCNCPoint5[11797] = {X 75.2381, Y 71.0959, Z -7.1667, A 0.000, B 0.000, C 0.000 }
gfCNCPoint5[11798] = {X 72.9995, Y 71.3838, Z -7.1667, A 0.000, B 0.000, C 0.000 }
gfCNCPoint5[11799] = {X 70.7445, Y 71.4800, Z -7.1667, A 0.000, B 0.000, C 0.000 }
gfCNCPoint5[11800] = {X 64.1851, Y 71.4800, Z -7.1667, A 0.000, B 0.000, C 0.000 }
gfCNCPoint5[11801] = {X 62.0752, Y 71.3958, Z -7.1667, A 0.000, B 0.000, C 0.000 }
gfCNCPoint5[11802] = {X 59.9787, Y 71.1438, Z -7.1667, A 0.000, B 0.000, C 0.000 }
gfCNCPoint5[11803] = {X 57.9089, Y 70.7255, Z -7.1667, A 0.000, B 0.000, C 0.000 }
gfCNCPoint5[11804] = {X 55.8790, Y 70.1436, Z -7.1667, A 0.000, B 0.000, C 0.000 }
gfCNCPoint5[11805] = {X 53.8492, Y 70.7255, Z -7.1667, A 0.000, B 0.000, C 0.000 }
gfCNCPoint5[11806] = {X 51.7794, Y 71.1438, Z -7.1667, A 0.000, B 0.000, C 0.000 }
gfCNCPoint5[11807] = {X 49.6829, Y 71.3958, Z -7.1667, A 0.000, B 0.000, C 0.000 }
gfCNCPoint5[11808] = {X 47.5729, Y 71.4800, Z -7.1667, A 0.000, B 0.000, C 0.000 }
gfCNCPoint5[11809] = {X 40.6393, Y 71.4800, Z -7.1667, A 0.000, B 0.000, C 0.000 }
gfCNCPoint5[11810] = {X 38.8059, Y 71.4165, Z -7.1667, A 0.000, B 0.000, C 0.000 }
gfCNCPoint5[11811] = {X 36.9813, Y 71.2261, Z -7.1667, A 0.000, B 0.000, C 0.000 }
gfCNCPoint5[11812] = {X 34.4004, Y 72.0356, Z -7.1667, A 0.000, B 0.000, C 0.000 }
gfCNCPoint5[11813] = {X 31.7586, Y 72.6157, Z -7.1667, A 0.000, B 0.000, C 0.000 }
gfCNCPoint5[11814] = {X 30.3337, Y 73.1751, Z -7.1667, A 0.000, B 0.000, C 0.000 }
gfCNCPoint5[11815] = {X 28.8941, Y 73.6951, Z -7.1667, A 0.000, B 0.000, C 0.000 }
gfCNCPoint5[11816] = {X 108.0295, Y 73.6951, Z -7.1667, A 0.000, B 0.000, C 0.000 }
gfCNCPoint5[11817] = {X 110.0244, Y 72.3689, Z -7.1667, A 0.000, B 0.000, C 0.000 }
gfCNCPoint5[11818] = {X 112.1224, Y 71.2125, Z -7.1667, A 0.000, B 0.000, C 0.000 }
gfCNCPoint5[11819] = {X 113.1243, Y 70.7371, Z -7.1667, A 0.000, B 0.000, C 0.000 }
gfCNCPoint5[11820] = {X 114.1437, Y 70.3005, Z -7.1667, A 0.000, B 0.000, C 0.000 }
gfCNCPoint5[11821] = {X 117.4408, Y 66.6800, Z -7.1667, A 0.000, B 0.000, C 0.000 }
gfCNCPoint5[11822] = {X 111.9185, Y 66.6800, Z -7.1667, A 0.000, B 0.000, C 0.000 }
gfCNCPoint5[11823] = {X 111.5284, Y 66.6765, Z -7.1667, A 0.000, B 0.000, C 0.000 }
gfCNCPoint5[11824] = {X 111.1384, Y 66.6660, Z -7.1667, A 0.000, B 0.000, C 0.000 }
gfCNCPoint5[11825] = {X 111.2248, Y 64.2675, Z -7.1667, A 0.000, B 0.000, C 0.000 }
gfCNCPoint5[11826] = {X 109.1059, Y 64.0737, Z -7.1667, A 0.000, B 0.000, C 0.000 }
gfCNCPoint5[11827] = {X 107.0213, Y 63.6477, Z -7.1667, A 0.000, B 0.000, C 0.000 }
gfCNCPoint5[11828] = {X 105.0841, Y 64.0514, Z -7.1667, A 0.000, B 0.000, C 0.000 }
gfCNCPoint5[11829] = {X 103.1158, Y 64.2545, Z -7.1667, A 0.000, B 0.000, C 0.000 }
gfCNCPoint5[11830] = {X 101.1370, Y 64.2547, Z -7.1667, A 0.000, B 0.000, C 0.000 }
gfCNCPoint5[11831] = {X 99.1686, Y 64.0521, Z -7.1667, A 0.000, B 0.000, C 0.000 }
gfCNCPoint5[11832] = {X 97.2313, Y 63.6488, Z -7.1667, A 0.000, B 0.000, C 0.000 }
gfCNCPoint5[11833] = {X 95.6204, Y 63.9986, Z -7.1667, A 0.000, B 0.000, C 0.000 }
gfCNCPoint5[11834] = {X 93.9855, Y 64.2095, Z -7.1667, A 0.000, B 0.000, C 0.000 }
gfCNCPoint5[11835] = {X 92.3385, Y 64.2800, Z -7.1667, A 0.000, B 0.000, C 0.000 }
gfCNCPoint5[11836] = {X 85.8951, Y 64.2800, Z -7.1667, A 0.000, B 0.000, C 0.000 }
gfCNCPoint5[11837] = {X 85.5417, Y 64.2768, Z -7.1667, A 0.000, B 0.000, C 0.000 }
gfCNCPoint5[11838] = {X 85.1884, Y 64.2670, Z -7.1667, A 0.000, B 0.000, C 0.000 }
gfCNCPoint5[11839] = {X 83.3593, Y 65.5113, Z -7.1667, A 0.000, B 0.000, C 0.000 }
gfCNCPoint5[11840] = {X 81.4238, Y 66.5824, Z -7.1667, A 0.000, B 0.000, C 0.000 }
gfCNCPoint5[11841] = {X 79.3981, Y 67.4713, Z -7.1667, A 0.000, B 0.000, C 0.000 }
gfCNCPoint5[11842] = {X 77.2994, Y 68.1706, Z -7.1667, A 0.000, B 0.000, C 0.000 }
gfCNCPoint5[11843] = {X 75.1454, Y 68.6744, Z -7.1667, A 0.000, B 0.000, C 0.000 }
gfCNCPoint5[11844] = {X 72.9543, Y 68.9784, Z -7.1667, A 0.000, B 0.000, C 0.000 }
gfCNCPoint5[11845] = {X 70.7445, Y 69.0800, Z -7.1667, A 0.000, B 0.000, C 0.000 }
gfCNCPoint5[11846] = {X 64.1851, Y 69.0800, Z -7.1667, A 0.000, B 0.000, C 0.000 }
gfCNCPoint5[11847] = {X 62.0678, Y 68.9867, Z -7.1667, A 0.000, B 0.000, C 0.000 }
gfCNCPoint5[11848] = {X 59.9669, Y 68.7076, Z -7.1667, A 0.000, B 0.000, C 0.000 }
gfCNCPoint5[11849] = {X 57.8986, Y 68.2449, Z -7.1667, A 0.000, B 0.000, C 0.000 }
gfCNCPoint5[11850] = {X 55.8790, Y 67.6021, Z -7.1667, A 0.000, B 0.000, C 0.000 }
gfCNCPoint5[11851] = {X 53.8595, Y 68.2449, Z -7.1667, A 0.000, B 0.000, C 0.000 }
gfCNCPoint5[11852] = {X 51.7912, Y 68.7076, Z -7.1667, A 0.000, B 0.000, C 0.000 }
gfCNCPoint5[11853] = {X 49.6903, Y 68.9867, Z -7.1667, A 0.000, B 0.000, C 0.000 }
gfCNCPoint5[11854] = {X 47.5729, Y 69.0800, Z -7.1667, A 0.000, B 0.000, C 0.000 }
gfCNCPoint5[11855] = {X 40.6393, Y 69.0800, Z -7.1667, A 0.000, B 0.000, C 0.000 }
gfCNCPoint5[11856] = {X 38.6753, Y 68.9998, Z -7.1667, A 0.000, B 0.000, C 0.000 }
gfCNCPoint5[11857] = {X 36.7244, Y 68.7596, Z -7.1667, A 0.000, B 0.000, C 0.000 }
gfCNCPoint5[11858] = {X 34.8840, Y 69.3996, Z -7.1667, A 0.000, B 0.000, C 0.000 }
gfCNCPoint5[11859] = {X 33.0040, Y 69.9119, Z -7.1667, A 0.000, B 0.000, C 0.000 }
gfCNCPoint5[11860] = {X 31.0934, Y 70.2941, Z -7.1667, A 0.000, B 0.000, C 0.000 }
gfCNCPoint5[11861] = {X 29.6101, Y 70.8829, Z -7.1667, A 0.000, B 0.000, C 0.000 }
gfCNCPoint5[11862] = {X 28.1098, Y 71.4269, Z -7.1667, A 0.000, B 0.000, C 0.000 }
gfCNCPoint5[11863] = {X 27.6086, Y 71.5974, Z -7.1667, A 0.000, B 0.000, C 0.000 }
gfCNCPoint5[11864] = {X 27.1057, Y 71.7629, Z -7.1667, A 0.000, B 0.000, C 0.000 }
gfCNCPoint5[11865] = {X 25.5128, Y 72.2546, Z -7.1667, A 0.000, B 0.000, C 0.000 }
gfCNCPoint5[11866] = {X 23.9033, Y 72.6893, Z -7.1667, A 0.000, B 0.000, C 0.000 }
gfCNCPoint5[11867] = {X 23.9033, Y 76.0951, Z -7.1667, A 0.000, B 0.000, C 0.000 }
gfCNCPoint5[11868] = {X 108.8280, Y 76.0951, Z -7.1667, A 0.000, B 0.000, C 0.000 }
gfCNCPoint5[11869] = {X 110.3990, Y 74.9721, Z -7.1667, A 0.000, B 0.000, C 0.000 }
gfCNCPoint5[11870] = {X 112.0477, Y 73.9666, Z -7.1667, A 0.000, B 0.000, C 0.000 }
gfCNCPoint5[11871] = {X 113.7653, Y 73.0839, Z -7.1667, A 0.000, B 0.000, C 0.000 }
gfCNCPoint5[11872] = {X 115.5427, Y 72.3287, Z -7.1667, A 0.000, B 0.000, C 0.000 }
gfCNCPoint5[11873] = {X 123.7246, Y 63.3444, Z -7.1667, A 0.000, B 0.000, C 0.000 }
gfCNCPoint5[11874] = {X 121.7831, Y 63.8623, Z -7.1667, A 0.000, B 0.000, C 0.000 }
gfCNCPoint5[11875] = {X 119.7982, Y 64.1753, Z -7.1667, A 0.000, B 0.000, C 0.000 }
gfCNCPoint5[11876] = {X 117.7916, Y 64.2800, Z -7.1667, A 0.000, B 0.000, C 0.000 }
gfCNCPoint5[11877] = {X 111.9185, Y 64.2800, Z -7.1667, A 0.000, B 0.000, C 0.000 }
gfCNCPoint5[11878] = {X 111.5716, Y 64.2769, Z -7.1667, A 0.000, B 0.000, C 0.000 }
gfCNCPoint5[11879] = {X 111.2248, Y 64.2675, Z -7.1667, A 0.000, B 0.000, C 0.000 }
gfCNCPoint5[11880] = {X 111.3111, Y 61.8691, Z -7.1667, A 0.000, B 0.000, C 0.000 }
gfCNCPoint5[11881] = {X 109.8624, Y 61.7543, Z -7.1667, A 0.000, B 0.000, C 0.000 }
gfCNCPoint5[11882] = {X 108.4289, Y 61.5154, Z -7.1667, A 0.000, B 0.000, C 0.000 }
gfCNCPoint5[11883] = {X 107.0213, Y 61.1540, Z -7.1667, A 0.000, B 0.000, C 0.000 }
gfCNCPoint5[11884] = {X 105.0907, Y 61.6173, Z -7.1667, A 0.000, B 0.000, C 0.000 }
gfCNCPoint5[11885] = {X 103.1191, Y 61.8506, Z -7.1667, A 0.000, B 0.000, C 0.000 }
gfCNCPoint5[11886] = {X 101.1337, Y 61.8509, Z -7.1667, A 0.000, B 0.000, C 0.000 }
gfCNCPoint5[11887] = {X 99.1620, Y 61.6181, Z -7.1667, A 0.000, B 0.000, C 0.000 }
gfCNCPoint5[11888] = {X 97.2313, Y 61.1553, Z -7.1667, A 0.000, B 0.000, C 0.000 }
gfCNCPoint5[11889] = {X 95.6267, Y 61.5566, Z -7.1667, A 0.000, B 0.000, C 0.000 }
gfCNCPoint5[11890] = {X 93.9906, Y 61.7990, Z -7.1667, A 0.000, B 0.000, C 0.000 }
gfCNCPoint5[11891] = {X 92.3385, Y 61.8800, Z -7.1667, A 0.000, B 0.000, C 0.000 }
gfCNCPoint5[11892] = {X 85.8951, Y 61.8800, Z -7.1667, A 0.000, B 0.000, C 0.000 }
gfCNCPoint5[11893] = {X 85.1609, Y 61.8640, Z -7.1667, A 0.000, B 0.000, C 0.000 }
gfCNCPoint5[11894] = {X 84.4280, Y 61.8161, Z -7.1667, A 0.000, B 0.000, C 0.000 }
gfCNCPoint5[11895] = {X 82.7247, Y 63.0692, Z -7.1667, A 0.000, B 0.000, C 0.000 }
gfCNCPoint5[11896] = {X 80.9073, Y 64.1504, Z -7.1667, A 0.000, B 0.000, C 0.000 }
gfCNCPoint5[11897] = {X 78.9932, Y 65.0494, Z -7.1667, A 0.000, B 0.000, C 0.000 }
gfCNCPoint5[11898] = {X 77.0007, Y 65.7577, Z -7.1667, A 0.000, B 0.000, C 0.000 }
gfCNCPoint5[11899] = {X 74.9487, Y 66.2685, Z -7.1667, A 0.000, B 0.000, C 0.000 }
gfCNCPoint5[11900] = {X 72.8566, Y 66.5769, Z -7.1667, A 0.000, B 0.000, C 0.000 }
gfCNCPoint5[11901] = {X 70.7445, Y 66.6800, Z -7.1667, A 0.000, B 0.000, C 0.000 }
gfCNCPoint5[11902] = {X 64.1851, Y 66.6800, Z -7.1667, A 0.000, B 0.000, C 0.000 }
gfCNCPoint5[11903] = {X 62.0576, Y 66.5754, Z -7.1667, A 0.000, B 0.000, C 0.000 }
gfCNCPoint5[11904] = {X 59.9505, Y 66.2624, Z -7.1667, A 0.000, B 0.000, C 0.000 }
gfCNCPoint5[11905] = {X 57.8844, Y 65.7442, Z -7.1667, A 0.000, B 0.000, C 0.000 }
gfCNCPoint5[11906] = {X 55.8790, Y 65.0258, Z -7.1667, A 0.000, B 0.000, C 0.000 }
gfCNCPoint5[11907] = {X 53.8737, Y 65.7442, Z -7.1667, A 0.000, B 0.000, C 0.000 }
gfCNCPoint5[11908] = {X 51.8075, Y 66.2624, Z -7.1667, A 0.000, B 0.000, C 0.000 }
gfCNCPoint5[11909] = {X 49.7005, Y 66.5753, Z -7.1667, A 0.000, B 0.000, C 0.000 }
gfCNCPoint5[11910] = {X 47.5729, Y 66.6800, Z -7.1667, A 0.000, B 0.000, C 0.000 }
gfCNCPoint5[11911] = {X 40.6393, Y 66.6800, Z -7.1667, A 0.000, B 0.000, C 0.000 }
gfCNCPoint5[11912] = {X 38.5453, Y 66.5786, Z -7.1667, A 0.000, B 0.000, C 0.000 }
gfCNCPoint5[11913] = {X 36.4710, Y 66.2755, Z -7.1667, A 0.000, B 0.000, C 0.000 }
gfCNCPoint5[11914] = {X 34.5060, Y 67.0017, Z -7.1667, A 0.000, B 0.000, C 0.000 }
gfCNCPoint5[11915] = {X 32.4890, Y 67.5675, Z -7.1667, A 0.000, B 0.000, C 0.000 }
gfCNCPoint5[11916] = {X 30.4330, Y 67.9691, Z -7.1667, A 0.000, B 0.000, C 0.000 }
gfCNCPoint5[11917] = {X 28.4136, Y 68.7685, Z -7.1667, A 0.000, B 0.000, C 0.000 }
gfCNCPoint5[11918] = {X 26.3619, Y 69.4811, Z -7.1667, A 0.000, B 0.000, C 0.000 }
gfCNCPoint5[11919] = {X 23.9510, Y 70.1979, Z -7.1667, A 0.000, B 0.000, C 0.000 }
gfCNCPoint5[11920] = {X 21.5033, Y 70.7771, Z -7.1667, A 0.000, B 0.000, C 0.000 }
gfCNCPoint5[11921] = {X 21.5033, Y 78.4951, Z -7.1667, A 0.000, B 0.000, C 0.000 }
gfCNCPoint5[11922] = {X 109.6679, Y 78.4951, Z -7.1667, A 0.000, B 0.000, C 0.000 }
gfCNCPoint5[11923] = {X 111.3402, Y 77.2322, Z -7.1667, A 0.000, B 0.000, C 0.000 }
gfCNCPoint5[11924] = {X 113.1159, Y 76.1195, Z -7.1667, A 0.000, B 0.000, C 0.000 }
gfCNCPoint5[11925] = {X 114.9817, Y 75.1654, Z -7.1667, A 0.000, B 0.000, C 0.000 }
gfCNCPoint5[11926] = {X 116.9233, Y 74.3771, Z -7.1667, A 0.000, B 0.000, C 0.000 }
gfCNCPoint5[11927] = {X 130.4102, Y 59.5676, Z -7.1667, A 0.000, B 0.000, C 0.000 }
gfCNCPoint5[11928] = {X 129.5273, Y 58.7527, Z -7.1667, A 0.000, B 0.000, C 0.000 }
gfCNCPoint5[11929] = {X 128.6970, Y 57.8844, Z -7.1667, A 0.000, B 0.000, C 0.000 }
gfCNCPoint5[11930] = {X 127.3923, Y 58.8838, Z -7.1667, A 0.000, B 0.000, C 0.000 }
gfCNCPoint5[11931] = {X 125.9967, Y 59.7516, Z -7.1667, A 0.000, B 0.000, C 0.000 }
gfCNCPoint5[11932] = {X 124.5233, Y 60.4796, Z -7.1667, A 0.000, B 0.000, C 0.000 }
gfCNCPoint5[11933] = {X 122.9860, Y 61.0609, Z -7.1667, A 0.000, B 0.000, C 0.000 }
gfCNCPoint5[11934] = {X 121.2862, Y 61.5143, Z -7.1667, A 0.000, B 0.000, C 0.000 }
gfCNCPoint5[11935] = {X 119.5484, Y 61.7883, Z -7.1667, A 0.000, B 0.000, C 0.000 }
gfCNCPoint5[11936] = {X 117.7916, Y 61.8800, Z -7.1667, A 0.000, B 0.000, C 0.000 }
gfCNCPoint5[11937] = {X 111.9185, Y 61.8800, Z -7.1667, A 0.000, B 0.000, C 0.000 }
gfCNCPoint5[11938] = {X 111.6148, Y 61.8773, Z -7.1667, A 0.000, B 0.000, C 0.000 }
gfCNCPoint5[11939] = {X 111.3111, Y 61.8691, Z -7.1667, A 0.000, B 0.000, C 0.000 }
gfCNCPoint5[11940] = {X 111.3975, Y 59.4706, Z -7.1667, A 0.000, B 0.000, C 0.000 }
gfCNCPoint5[11941] = {X 109.9123, Y 59.3403, Z -7.1667, A 0.000, B 0.000, C 0.000 }
gfCNCPoint5[11942] = {X 108.4484, Y 59.0581, Z -7.1667, A 0.000, B 0.000, C 0.000 }
gfCNCPoint5[11943] = {X 107.0213, Y 58.6267, Z -7.1667, A 0.000, B 0.000, C 0.000 }
gfCNCPoint5[11944] = {X 105.4260, Y 59.0985, Z -7.1667, A 0.000, B 0.000, C 0.000 }
gfCNCPoint5[11945] = {X 103.7872, Y 59.3842, Z -7.1667, A 0.000, B 0.000, C 0.000 }
gfCNCPoint5[11946] = {X 102.1264, Y 59.4800, Z -7.1667, A 0.000, B 0.000, C 0.000 }
gfCNCPoint5[11947] = {X 100.4656, Y 59.3847, Z -7.1667, A 0.000, B 0.000, C 0.000 }
gfCNCPoint5[11948] = {X 98.8267, Y 59.0996, Z -7.1667, A 0.000, B 0.000, C 0.000 }
gfCNCPoint5[11949] = {X 97.2313, Y 58.6283, Z -7.1667, A 0.000, B 0.000, C 0.000 }
gfCNCPoint5[11950] = {X 95.6367, Y 59.0994, Z -7.1667, A 0.000, B 0.000, C 0.000 }
gfCNCPoint5[11951] = {X 93.9986, Y 59.3845, Z -7.1667, A 0.000, B 0.000, C 0.000 }
gfCNCPoint5[11952] = {X 92.3385, Y 59.4800, Z -7.1667, A 0.000, B 0.000, C 0.000 }
gfCNCPoint5[11953] = {X 85.8951, Y 59.4800, Z -7.1667, A 0.000, B 0.000, C 0.000 }
gfCNCPoint5[11954] = {X 84.7780, Y 59.4368, Z -7.1667, A 0.000, B 0.000, C 0.000 }
gfCNCPoint5[11955] = {X 83.6677, Y 59.3077, Z -7.1667, A 0.000, B 0.000, C 0.000 }
gfCNCPoint5[11956] = {X 82.0978, Y 60.5827, Z -7.1667, A 0.000, B 0.000, C 0.000 }
gfCNCPoint5[11957] = {X 80.4031, Y 61.6862, Z -7.1667, A 0.000, B 0.000, C 0.000 }
gfCNCPoint5[11958] = {X 78.6021, Y 62.6061, Z -7.1667, A 0.000, B 0.000, C 0.000 }
gfCNCPoint5[11959] = {X 76.7146, Y 63.3324, Z -7.1667, A 0.000, B 0.000, C 0.000 }
gfCNCPoint5[11960] = {X 74.7614, Y 63.8569, Z -7.1667, A 0.000, B 0.000, C 0.000 }
gfCNCPoint5[11961] = {X 72.7640, Y 64.1739, Z -7.1667, A 0.000, B 0.000, C 0.000 }
gfCNCPoint5[11962] = {X 70.7445, Y 64.2800, Z -7.1667, A 0.000, B 0.000, C 0.000 }
gfCNCPoint5[11963] = {X 64.1851, Y 64.2800, Z -7.1667, A 0.000, B 0.000, C 0.000 }
gfCNCPoint5[11964] = {X 62.0428, Y 64.1606, Z -7.1667, A 0.000, B 0.000, C 0.000 }
gfCNCPoint5[11965] = {X 59.9269, Y 63.8039, Z -7.1667, A 0.000, B 0.000, C 0.000 }
gfCNCPoint5[11966] = {X 57.8638, Y 63.2143, Z -7.1667, A 0.000, B 0.000, C 0.000 }
gfCNCPoint5[11967] = {X 55.8790, Y 62.3991, Z -7.1667, A 0.000, B 0.000, C 0.000 }
gfCNCPoint5[11968] = {X 53.8942, Y 63.2143, Z -7.1667, A 0.000, B 0.000, C 0.000 }
gfCNCPoint5[11969] = {X 51.8311, Y 63.8039, Z -7.1667, A 0.000, B 0.000, C 0.000 }
gfCNCPoint5[11970] = {X 49.7153, Y 64.1606, Z -7.1667, A 0.000, B 0.000, C 0.000 }
gfCNCPoint5[11971] = {X 47.5729, Y 64.2800, Z -7.1667, A 0.000, B 0.000, C 0.000 }
gfCNCPoint5[11972] = {X 40.6393, Y 64.2800, Z -7.1667, A 0.000, B 0.000, C 0.000 }
gfCNCPoint5[11973] = {X 39.1552, Y 64.2228, Z -7.1667, A 0.000, B 0.000, C 0.000 }
gfCNCPoint5[11974] = {X 37.6799, Y 64.0515, Z -7.1667, A 0.000, B 0.000, C 0.000 }
gfCNCPoint5[11975] = {X 36.2222, Y 63.7672, Z -7.1667, A 0.000, B 0.000, C 0.000 }
gfCNCPoint5[11976] = {X 34.1369, Y 64.5949, Z -7.1667, A 0.000, B 0.000, C 0.000 }
gfCNCPoint5[11977] = {X 31.9825, Y 65.2210, Z -7.1667, A 0.000, B 0.000, C 0.000 }
gfCNCPoint5[11978] = {X 29.7784, Y 65.6397, Z -7.1667, A 0.000, B 0.000, C 0.000 }
gfCNCPoint5[11979] = {X 27.7161, Y 66.4672, Z -7.1667, A 0.000, B 0.000, C 0.000 }
gfCNCPoint5[11980] = {X 25.6181, Y 67.1993, Z -7.1667, A 0.000, B 0.000, C 0.000 }
gfCNCPoint5[11981] = {X 23.4755, Y 67.8405, Z -7.1667, A 0.000, B 0.000, C 0.000 }
gfCNCPoint5[11982] = {X 21.3019, Y 68.3669, Z -7.1667, A 0.000, B 0.000, C 0.000 }
gfCNCPoint5[11983] = {X 19.1033, Y 68.7770, Z -7.1667, A 0.000, B 0.000, C 0.000 }
gfCNCPoint5[11984] = {X 19.1033, Y 80.8951, Z -7.1667, A 0.000, B 0.000, C 0.000 }
gfCNCPoint5[11985] = {X 110.5566, Y 80.8951, Z -7.1667, A 0.000, B 0.000, C 0.000 }
gfCNCPoint5[11986] = {X 112.3046, Y 79.4889, Z -7.1667, A 0.000, B 0.000, C 0.000 }
gfCNCPoint5[11987] = {X 114.1886, Y 78.2708, Z -7.1667, A 0.000, B 0.000, C 0.000 }
gfCNCPoint5[11988] = {X 116.1883, Y 77.2539, Z -7.1667, A 0.000, B 0.000, C 0.000 }
gfCNCPoint5[11989] = {X 118.2824, Y 76.4491, Z -7.1667, A 0.000, B 0.000, C 0.000 }
gfCNCPoint5[11990] = {X 133.9623, Y 59.2315, Z -7.1667, A 0.000, B 0.000, C 0.000 }
gfCNCPoint5[11991] = {X 132.7149, Y 58.3542, Z -7.1667, A 0.000, B 0.000, C 0.000 }
gfCNCPoint5[11992] = {X 131.5517, Y 57.3678, Z -7.1667, A 0.000, B 0.000, C 0.000 }
gfCNCPoint5[11993] = {X 130.4824, Y 56.2805, Z -7.1667, A 0.000, B 0.000, C 0.000 }
gfCNCPoint5[11994] = {X 129.6655, Y 55.2988, Z -7.1667, A 0.000, B 0.000, C 0.000 }
gfCNCPoint5[11995] = {X 128.9251, Y 54.2582, Z -7.1667, A 0.000, B 0.000, C 0.000 }
gfCNCPoint5[11996] = {X 128.0750, Y 55.1942, Z -7.1667, A 0.000, B 0.000, C 0.000 }
gfCNCPoint5[11997] = {X 127.1464, Y 56.0525, Z -7.1667, A 0.000, B 0.000, C 0.000 }
gfCNCPoint5[11998] = {X 125.7915, Y 57.0695, Z -7.1667, A 0.000, B 0.000, C 0.000 }
gfCNCPoint5[11999] = {X 124.3270, Y 57.9212, Z -7.1667, A 0.000, B 0.000, C 0.000 }
gfCNCPoint5[12000] = {X 122.7731, Y 58.5961, Z -7.1667, A 0.000, B 0.000, C 0.000 }
gfCNCPoint5[12001] = {X 121.1510, Y 59.0849, Z -7.1667, A 0.000, B 0.000, C 0.000 }
gfCNCPoint5[12002] = {X 119.4828, Y 59.3809, Z -7.1667, A 0.000, B 0.000, C 0.000 }
gfCNCPoint5[12003] = {X 117.7916, Y 59.4800, Z -7.1667, A 0.000, B 0.000, C 0.000 }
gfCNCPoint5[12004] = {X 111.9185, Y 59.4800, Z -7.1667, A 0.000, B 0.000, C 0.000 }
gfCNCPoint5[12005] = {X 111.6579, Y 59.4777, Z -7.1667, A 0.000, B 0.000, C 0.000 }
gfCNCPoint5[12006] = {X 111.3975, Y 59.4706, Z -7.1667, A 0.000, B 0.000, C 0.000 }
gfCNCPoint5[12007] = {X 111.4838, Y 57.0722, Z -7.1667, A 0.000, B 0.000, C 0.000 }
gfCNCPoint5[12008] = {X 109.9566, Y 56.9196, Z -7.1667, A 0.000, B 0.000, C 0.000 }
gfCNCPoint5[12009] = {X 108.4610, Y 56.5746, Z -7.1667, A 0.000, B 0.000, C 0.000 }
gfCNCPoint5[12010] = {X 107.0213, Y 56.0428, Z -7.1667, A 0.000, B 0.000, C 0.000 }
gfCNCPoint5[12011] = {X 105.4432, Y 56.6151, Z -7.1667, A 0.000, B 0.000, C 0.000 }
gfCNCPoint5[12012] = {X 103.8010, Y 56.9630, Z -7.1667, A 0.000, B 0.000, C 0.000 }
gfCNCPoint5[12013] = {X 102.1265, Y 57.0800, Z -7.1667, A 0.000, B 0.000, C 0.000 }
gfCNCPoint5[12014] = {X 100.4519, Y 56.9637, Z -7.1667, A 0.000, B 0.000, C 0.000 }
gfCNCPoint5[12015] = {X 98.8096, Y 56.6164, Z -7.1667, A 0.000, B 0.000, C 0.000 }
gfCNCPoint5[12016] = {X 97.2313, Y 56.0448, Z -7.1667, A 0.000, B 0.000, C 0.000 }
gfCNCPoint5[12017] = {X 95.6538, Y 56.6162, Z -7.1667, A 0.000, B 0.000, C 0.000 }
gfCNCPoint5[12018] = {X 94.0123, Y 56.9635, Z -7.1667, A 0.000, B 0.000, C 0.000 }
gfCNCPoint5[12019] = {X 92.3385, Y 57.0800, Z -7.1667, A 0.000, B 0.000, C 0.000 }
gfCNCPoint5[12020] = {X 85.8951, Y 57.0800, Z -7.1667, A 0.000, B 0.000, C 0.000 }
gfCNCPoint5[12021] = {X 84.3894, Y 56.9858, Z -7.1667, A 0.000, B 0.000, C 0.000 }
gfCNCPoint5[12022] = {X 82.9073, Y 56.7047, Z -7.1667, A 0.000, B 0.000, C 0.000 }
gfCNCPoint5[12023] = {X 81.4846, Y 58.0224, Z -7.1667, A 0.000, B 0.000, C 0.000 }
gfCNCPoint5[12024] = {X 79.9203, Y 59.1682, Z -7.1667, A 0.000, B 0.000, C 0.000 }
gfCNCPoint5[12025] = {X 78.2348, Y 60.1271, Z -7.1667, A 0.000, B 0.000, C 0.000 }
gfCNCPoint5[12026] = {X 76.4504, Y 60.8863, Z -7.1667, A 0.000, B 0.000, C 0.000 }
gfCNCPoint5[12027] = {X 74.5908, Y 61.4359, Z -7.1667, A 0.000, B 0.000, C 0.000 }
gfCNCPoint5[12028] = {X 72.6804, Y 61.7686, Z -7.1667, A 0.000, B 0.000, C 0.000 }
gfCNCPoint5[12029] = {X 70.7445, Y 61.8800, Z -7.1667, A 0.000, B 0.000, C 0.000 }
gfCNCPoint5[12030] = {X 64.1851, Y 61.8800, Z -7.1667, A 0.000, B 0.000, C 0.000 }
gfCNCPoint5[12031] = {X 62.4514, Y 61.7907, Z -7.1667, A 0.000, B 0.000, C 0.000 }
gfCNCPoint5[12032] = {X 60.7359, Y 61.5238, Z -7.1667, A 0.000, B 0.000, C 0.000 }
gfCNCPoint5[12033] = {X 59.0570, Y 61.0822, Z -7.1667, A 0.000, B 0.000, C 0.000 }
gfCNCPoint5[12034] = {X 57.4323, Y 60.4704, Z -7.1667, A 0.000, B 0.000, C 0.000 }
gfCNCPoint5[12035] = {X 55.8790, Y 59.6950, Z -7.1667, A 0.000, B 0.000, C 0.000 }
gfCNCPoint5[12036] = {X 54.3258, Y 60.4704, Z -7.1667, A 0.000, B 0.000, C 0.000 }
gfCNCPoint5[12037] = {X 52.7011, Y 61.0822, Z -7.1667, A 0.000, B 0.000, C 0.000 }
gfCNCPoint5[12038] = {X 51.0221, Y 61.5238, Z -7.1667, A 0.000, B 0.000, C 0.000 }
gfCNCPoint5[12039] = {X 49.3067, Y 61.7907, Z -7.1667, A 0.000, B 0.000, C 0.000 }
gfCNCPoint5[12040] = {X 47.5729, Y 61.8800, Z -7.1667, A 0.000, B 0.000, C 0.000 }
gfCNCPoint5[12041] = {X 40.6393, Y 61.8800, Z -7.1667, A 0.000, B 0.000, C 0.000 }
gfCNCPoint5[12042] = {X 39.0681, Y 61.8067, Z -7.1667, A 0.000, B 0.000, C 0.000 }
gfCNCPoint5[12043] = {X 37.5105, Y 61.5875, Z -7.1667, A 0.000, B 0.000, C 0.000 }
gfCNCPoint5[12044] = {X 35.9801, Y 61.2243, Z -7.1667, A 0.000, B 0.000, C 0.000 }
gfCNCPoint5[12045] = {X 34.3403, Y 61.9607, Z -7.1667, A 0.000, B 0.000, C 0.000 }
gfCNCPoint5[12046] = {X 32.6440, Y 62.5556, Z -7.1667, A 0.000, B 0.000, C 0.000 }
gfCNCPoint5[12047] = {X 30.9034, Y 63.0048, Z -7.1667, A 0.000, B 0.000, C 0.000 }
gfCNCPoint5[12048] = {X 29.1310, Y 63.3049, Z -7.1667, A 0.000, B 0.000, C 0.000 }
gfCNCPoint5[12049] = {X 27.0225, Y 64.1638, Z -7.1667, A 0.000, B 0.000, C 0.000 }
gfCNCPoint5[12050] = {X 24.8742, Y 64.9175, Z -7.1667, A 0.000, B 0.000, C 0.000 }
gfCNCPoint5[12051] = {X 22.1942, Y 65.6949, Z -7.1667, A 0.000, B 0.000, C 0.000 }
gfCNCPoint5[12052] = {X 19.4660, Y 66.2819, Z -7.1667, A 0.000, B 0.000, C 0.000 }
gfCNCPoint5[12053] = {X 16.7033, Y 66.6755, Z -7.1667, A 0.000, B 0.000, C 0.000 }
gfCNCPoint5[12054] = {X 16.7033, Y 83.2951, Z -7.1667, A 0.000, B 0.000, C 0.000 }
gfCNCPoint5[12055] = {X 111.5037, Y 83.2951, Z -7.1667, A 0.000, B 0.000, C 0.000 }
gfCNCPoint5[12056] = {X 112.9228, Y 82.0345, Z -7.1667, A 0.000, B 0.000, C 0.000 }
gfCNCPoint5[12057] = {X 114.4589, Y 80.9196, Z -7.1667, A 0.000, B 0.000, C 0.000 }
